  MoveL 1328 to (313.05, 55, -156.48) mm, rotated rx -179.9 ry 0 rz -90 deg; joints [36.817, -66.564, 102.365, -127.219, 48.796, 139.976]
  MoveL 1329 to (313.57, 54.92, -158.6) mm, rotated rx -179.9 ry 0 rz -90 deg; joints [36.783, -66.439, 102.192, -127.22, 48.744, 139.947]
  MoveL 1330 to (314.82, 54.85, -160.4) mm, rotated rx -179.9 ry 0 rz -90 deg; joints [36.779, -66.303, 102.002, -127.186, 48.71, 139.892]
  MoveL 1331 to (316.62, 54.77, -161.63) mm, rotated rx -179.9 ry 0 rz -90 deg; joints [36.807, -66.175, 101.822, -127.121, 48.697, 139.819]
  MoveL 1332 to (318.74, 54.69, -162.14) mm, rotated rx -179.9 ry 0 rz -90 deg; joints [36.863, -66.07, 101.676, -127.036, 48.707, 139.738]
  MoveL 1333 to (320.91, 54.62, -161.86) mm, rotated rx -179.9 ry 0 rz -90 deg; joints [36.938, -66.003, 101.582, -126.941, 48.74, 139.661]
  MoveL 1334 to (322.84, 54.54, -160.83) mm, rotated rx -179.9 ry 0 rz -90 deg; joints [37.023, -65.981, 101.554, -126.851, 48.792, 139.599]
  MoveL 1335 to (324.27, 54.46, -159.18) mm, rotated rx -179.9 ry 0 rz -90 deg; joints [37.108, -66.007, 101.595, -126.776, 48.857, 139.561]
  MoveL 1336 to (325.02, 54.39, -157.13) mm, rotated rx -179.9 ry 0 rz -90 deg; joints [37.181, -66.077, 101.702, -126.728, 48.925, 139.552]
  MoveL 1337 to (324.98, 54.31, -154.94) mm, rotated rx -179.9 ry 0 rz -90 deg; joints [37.232, -66.183, 101.859, -126.712, 48.99, 139.573]
  MoveL 1338 to (324.18, 54.23, -152.91) mm, rotated rx -179.9 ry 0 rz -90 deg; joints [37.256, -66.31, 102.047, -126.731, 49.042, 139.623]
  MoveL 1339 to (322.7, 54.16, -151.3) mm, rotated rx -179.9 ry 0 rz -90 deg; joints [37.248, -66.44, 102.241, -126.783, 49.075, 139.696]
  MoveL 1340 to (320.75, 54.08, -150.32) mm, rotated rx -179.9 ry 0 rz -90 deg; joints [37.21, -66.557, 102.416, -126.862, 49.085, 139.782]
  MoveL 1341 to (318.57, 54, -150.11) mm, rotated rx -179.9 ry 0 rz -90 deg; joints [37.146, -66.646, 102.55, -126.958, 49.071, 139.872]
  MoveL 1342 to (316.46, 53.93, -150.68) mm, rotated rx -179.9 ry 0 rz -90 deg; joints [37.065, -66.693, 102.626, -127.059, 49.036, 139.954]
  MoveL 1343 to (314.7, 53.85, -151.96) mm, rotated rx -179.9 ry 0 rz -90 deg; joints [36.978, -66.692, 102.633, -127.153, 48.984, 140.018]
  MoveL 1344 to (313.5, 53.77, -153.79) mm, rotated rx -179.9 ry 0 rz -90 deg; joints [36.896, -66.644, 102.572, -127.226, 48.923, 140.058]
  MoveL 1345 to (313.04, 53.69, -155.93) mm, rotated rx -179.9 ry 0 rz -90 deg; joints [36.83, -66.554, 102.45, -127.271, 48.862, 140.067]
  MoveL 1346 to (313.37, 53.62, -158.09) mm, rotated rx -179.9 ry 0 rz -90 deg; joints [36.789, -66.434, 102.284, -127.281, 48.807, 140.045]
  MoveL 1347 to (314.44, 53.54, -159.99) mm, rotated rx -179.9 ry 0 rz -90 deg; joints [36.778, -66.299, 102.096, -127.255, 48.768, 139.996]
  MoveL 1348 to (316.12, 53.46, -161.38) mm, rotated rx -179.9 ry 0 rz -90 deg; joints [36.798, -66.168, 101.911, -127.198, 48.749, 139.927]
  MoveL 1349 to (318.19, 53.39, -162.09) mm, rotated rx -179.9 ry 0 rz -90 deg; joints [36.847, -66.056, 101.754, -127.116, 48.753, 139.847]
  MoveL 1350 to (320.38, 53.31, -162.01) mm, rotated rx -179.9 ry 0 rz -90 deg; joints [36.918, -65.978, 101.646, -127.023, 48.781, 139.768]
  MoveL 1351 to (322.39, 53.23, -161.15) mm, rotated rx -179.9 ry 0 rz -90 deg; joints [37.002, -65.944, 101.6, -126.93, 48.828, 139.702]
  MoveL 1352 to (323.96, 53.16, -159.64) mm, rotated rx -179.9 ry 0 rz -90 deg; joints [37.088, -65.958, 101.624, -126.851, 48.89, 139.657]
  MoveL 1353 to (324.9, 53.08, -157.67) mm, rotated rx -179.9 ry 0 rz -90 deg; joints [37.165, -66.018, 101.715, -126.795, 48.959, 139.64]
  MoveL 1354 to (325.07, 53, -155.49) mm, rotated rx -179.9 ry 0 rz -90 deg; joints [37.222, -66.116, 101.861, -126.77, 49.025, 139.654]
  MoveL 1355 to (324.45, 52.93, -153.39) mm, rotated rx -179.9 ry 0 rz -90 deg; joints [37.253, -66.239, 102.044, -126.78, 49.081, 139.697]
  MoveL 1356 to (323.13, 52.85, -151.65) mm, rotated rx -179.9 ry 0 rz -90 deg; joints [37.254, -66.37, 102.239, -126.824, 49.119, 139.764]
  MoveL 1357 to (321.27, 52.77, -150.5) mm, rotated rx -179.9 ry 0 rz -90 deg; joints [37.223, -66.492, 102.421, -126.897, 49.135, 139.848]
  MoveL 1358 to (319.13, 52.7, -150.09) mm, rotated rx -179.9 ry 0 rz -90 deg; joints [37.165, -66.589, 102.567, -126.99, 49.128, 139.938]
  MoveL 1359 to (316.97, 52.62, -150.46) mm, rotated rx -179.9 ry 0 rz -90 deg; joints [37.087, -66.647, 102.659, -127.091, 49.098, 140.023]
  MoveL 1360 to (315.1, 52.54, -151.58) mm, rotated rx -179.9 ry 0 rz -90 deg; joints [37.001, -66.659, 102.684, -127.188, 49.05, 140.093]
  MoveL 1361 to (313.74, 52.47, -153.29) mm, rotated rx -179.9 ry 0 rz -90 deg; joints [36.916, -66.622, 102.639, -127.268, 48.99, 140.139]
  MoveL 1362 to (313.08, 52.39, -155.37) mm, rotated rx -179.9 ry 0 rz -90 deg; joints [36.846, -66.542, 102.531, -127.321, 48.928, 140.156]
  MoveL 1363 to (313.21, 52.31, -157.56) mm, rotated rx -179.9 ry 0 rz -90 deg; joints [36.797, -66.428, 102.375, -127.34, 48.871, 140.142]
  MoveL 1364 to (314.11, 52.24, -159.55) mm, rotated rx -179.9 ry 0 rz -90 deg; joints [36.778, -66.296, 102.19, -127.323, 48.827, 140.099]
  MoveL 1365 to (315.65, 52.16, -161.09) mm, rotated rx -179.9 ry 0 rz -90 deg; joints [36.791, -66.162, 102.002, -127.273, 48.803, 140.034]
  MoveL 1366 to (317.65, 52.08, -161.98) mm, rotated rx -179.9 ry 0 rz -90 deg; joints [36.833, -66.043, 101.836, -127.196, 48.801, 139.956]
  MoveL 1367 to (319.83, 52.01, -162.1) mm, rotated rx -179.9 ry 0 rz -90 deg; joints [36.899, -65.956, 101.713, -127.105, 48.822, 139.876]
  MoveL 1368 to (321.91, 51.93, -161.44) mm, rotated rx -179.9 ry 0 rz -90 deg; joints [36.981, -65.91, 101.651, -127.011, 48.865, 139.805]
  MoveL 1369 to (323.62, 51.85, -160.08) mm, rotated rx -179.9 ry 0 rz -90 deg; joints [37.067, -65.912, 101.658, -126.926, 48.924, 139.754]
  MoveL 1370 to (324.73, 51.78, -158.2) mm, rotated rx -179.9 ry 0 rz -90 deg; joints [37.148, -65.961, 101.732, -126.864, 48.992, 139.729]
  MoveL 1371 to (325.1, 51.7, -156.04) mm, rotated rx -179.9 ry 0 rz -90 deg; joints [37.211, -66.05, 101.866, -126.831, 49.059, 139.735]
  MoveL 1372 to (324.68, 51.62, -153.9) mm, rotated rx -179.9 ry 0 rz -90 deg; joints [37.249, -66.168, 102.041, -126.832, 49.119, 139.772]
  MoveL 1373 to (323.52, 51.55, -152.05) mm, rotated rx -179.9 ry 0 rz -90 deg; joints [37.257, -66.299, 102.235, -126.868, 49.162, 139.834]
  MoveL 1374 to (321.78, 51.47, -150.73) mm, rotated rx -179.9 ry 0 rz -90 deg; joints [37.234, -66.425, 102.423, -126.934, 49.184, 139.914]
  MoveL 1375 to (319.68, 51.39, -150.12) mm, rotated rx -179.9 ry 0 rz -90 deg; joints [37.182, -66.529, 102.581, -127.023, 49.183, 140.004]
  MoveL 1376 to (317.5, 51.32, -150.29) mm, rotated rx -179.9 ry 0 rz -90 deg; joints [37.109, -66.598, 102.687, -127.123, 49.158, 140.091]
  MoveL 1377 to (315.53, 51.24, -151.23) mm, rotated rx -179.9 ry 0 rz -90 deg; joints [37.024, -66.622, 102.73, -127.222, 49.114, 140.165]
  MoveL 1378 to (314.02, 51.16, -152.81) mm, rotated rx -179.9 ry 0 rz -90 deg; joints [36.938, -66.597, 102.702, -127.307, 49.057, 140.218]
  MoveL 1379 to (313.18, 51.09, -154.83) mm, rotated rx -179.9 ry 0 rz -90 deg; joints [36.862, -66.528, 102.61, -127.368, 48.995, 140.243]
  MoveL 1380 to (313.1, 51.01, -157.01) mm, rotated rx -179.9 ry 0 rz -90 deg; joints [36.808, -66.421, 102.463, -127.396, 48.936, 140.236]
  MoveL 1381 to (313.81, 50.93, -159.08) mm, rotated rx -179.9 ry 0 rz -90 deg; joints [36.781, -66.292, 102.284, -127.388, 48.888, 140.2]
  MoveL 1382 to (315.21, 50.86, -160.76) mm, rotated rx -179.9 ry 0 rz -90 deg; joints [36.785, -66.157, 102.094, -127.346, 48.858, 140.14]
  MoveL 1383 to (317.12, 50.78, -161.83) mm, rotated rx -179.9 ry 0 rz -90 deg; joints [36.82, -66.033, 101.92, -127.275, 48.85, 140.064]
  MoveL 1384 to (319.28, 50.7, -162.15) mm, rotated rx -179.9 ry 0 rz -90 deg; joints [36.881, -65.936, 101.785, -127.186, 48.866, 139.983]
  MoveL 1385 to (321.41, 50.63, -161.68) mm, rotated rx -179.9 ry 0 rz -90 deg; joints [36.96, -65.879, 101.706, -127.091, 48.904, 139.909]
  MoveL 1386 to (323.24, 50.55, -160.48) mm, rotated rx -179.9 ry 0 rz -90 deg; joints [37.046, -65.869, 101.695, -127.004, 48.959, 139.852]
  MoveL 1387 to (324.52, 50.47, -158.71) mm, rotated rx -179.9 ry 0 rz -90 deg; joints [37.129, -65.907, 101.753, -126.934, 49.025, 139.821]
  MoveL 1388 to (325.08, 50.4, -156.59) mm, rotated rx -179.9 ry 0 rz -90 deg; joints [37.198, -65.987, 101.873, -126.893, 49.093, 139.819]
  MoveL 1389 to (324.86, 50.32, -154.42) mm, rotated rx -179.9 ry 0 rz -90 deg; joints [37.243, -66.099, 102.04, -126.885, 49.156, 139.848]
  MoveL 1390 to (323.87, 50.24, -152.47) mm, rotated rx -179.9 ry 0 rz -90 deg; joints [37.259, -66.228, 102.232, -126.913, 49.204, 139.904]
  MoveL 1391 to (322.26, 50.17, -151) mm, rotated rx -179.9 ry 0 rz -90 deg; joints [37.243, -66.356, 102.424, -126.972, 49.232, 139.981]
  MoveL 1392 to (320.23, 50.09, -150.2) mm, rotated rx -179.9 ry 0 rz -90 deg; joints [37.198, -66.467, 102.591, -127.056, 49.236, 140.069]
  MoveL 1393 to (318.04, 50.01, -150.17) mm, rotated rx -179.9 ry 0 rz -90 deg; joints [37.13, -66.546, 102.712, -127.154, 49.218, 140.158]
  MoveL 1394 to (315.99, 49.94, -150.93) mm, rotated rx -179.9 ry 0 rz -90 deg; joints [37.046, -66.582, 102.771, -127.255, 49.178, 140.236]
  MoveL 1395 to (314.35, 49.86, -152.36) mm, rotated rx -179.9 ry 0 rz -90 deg; joints [36.959, -66.57, 102.761, -127.345, 49.124, 140.295]
  MoveL 1396 to (313.32, 49.78, -154.29) mm, rotated rx -179.9 ry 0 rz -90 deg; joints [36.88, -66.511, 102.684, -127.413, 49.062, 140.327]
  MoveL 1397 to (313.05, 49.71, -156.46) mm, rotated rx -179.9 ry 0 rz -90 deg; joints [36.82, -66.412, 102.55, -127.449, 49.002, 140.329]
  MoveL 1398 to (313.56, 49.63, -158.58) mm, rotated rx -179.9 ry 0 rz -90 deg; joints [36.785, -66.287, 102.376, -127.451, 48.95, 140.3]
  MoveL 1399 to (314.8, 49.55, -160.38) mm, rotated rx -179.9 ry 0 rz -90 deg; joints [36.782, -66.152, 102.187, -127.417, 48.915, 140.245]
  MoveL 1400 to (316.6, 49.48, -161.62) mm, rotated rx -179.9 ry 0 rz -90 deg; joints [36.81, -66.024, 102.007, -127.352, 48.901, 140.172]
  MoveL 1401 to (318.72, 49.4, -162.14) mm, rotated rx -179.9 ry 0 rz -90 deg; joints [36.865, -65.919, 101.86, -127.267, 48.911, 140.091]
  MoveL 1402 to (320.89, 49.32, -161.87) mm, rotated rx -179.9 ry 0 rz -90 deg; joints [36.94, -65.851, 101.765, -127.173, 48.943, 140.015]
  MoveL 1403 to (322.82, 49.25, -160.84) mm, rotated rx -179.9 ry 0 rz -90 deg; joints [37.025, -65.829, 101.737, -127.082, 48.994, 139.953]
  MoveL 1404 to (324.26, 49.17, -159.19) mm, rotated rx -179.9 ry 0 rz -90 deg; joints [37.11, -65.855, 101.778, -127.007, 49.058, 139.914]
  MoveL 1405 to (325.01, 49.09, -157.14) mm, rotated rx -179.9 ry 0 rz -90 deg; joints [37.183, -65.925, 101.883, -126.958, 49.127, 139.905]
  MoveL 1406 to (324.99, 49.01, -154.96) mm, rotated rx -179.9 ry 0 rz -90 deg; joints [37.235, -66.03, 102.04, -126.941, 49.192, 139.926]
  MoveL 1407 to (324.19, 48.94, -152.93) mm, rotated rx -179.9 ry 0 rz -90 deg; joints [37.258, -66.156, 102.228, -126.96, 49.244, 139.976]
  MoveL 1408 to (322.72, 48.86, -151.31) mm, rotated rx -179.9 ry 0 rz -90 deg; joints [37.251, -66.286, 102.422, -127.011, 49.278, 140.048]
  MoveL 1409 to (320.76, 48.78, -150.33) mm, rotated rx -179.9 ry 0 rz -90 deg; joints [37.213, -66.403, 102.598, -127.09, 49.288, 140.134]
  MoveL 1410 to (318.59, 48.71, -150.1) mm, rotated rx -179.9 ry 0 rz -90 deg; joints [37.149, -66.492, 102.732, -127.186, 49.276, 140.224]
  MoveL 1411 to (316.48, 48.63, -150.67) mm, rotated rx -179.9 ry 0 rz -90 deg; joints [37.069, -66.539, 102.808, -127.287, 49.241, 140.306]
  MoveL 1412 to (314.71, 48.55, -151.95) mm, rotated rx -179.9 ry 0 rz -90 deg; joints [36.982, -66.539, 102.816, -127.381, 49.19, 140.37]
  MoveL 1413 to (313.51, 48.48, -153.77) mm, rotated rx -179.9 ry 0 rz -90 deg; joints [36.9, -66.491, 102.755, -127.455, 49.13, 140.41]
  MoveL 1414 to (313.04, 48.4, -155.91) mm, rotated rx -179.9 ry 0 rz -90 deg; joints [36.833, -66.402, 102.634, -127.5, 49.068, 140.419]
  MoveL 1415 to (313.36, 48.32, -158.07) mm, rotated rx -179.9 ry 0 rz -90 deg; joints [36.792, -66.282, 102.468, -127.511, 49.013, 140.398]
  MoveL 1416 to (314.43, 48.25, -159.97) mm, rotated rx -179.9 ry 0 rz -90 deg; joints [36.781, -66.148, 102.28, -127.485, 48.973, 140.349]
  MoveL 1417 to (316.11, 48.17, -161.37) mm, rotated rx -179.9 ry 0 rz -90 deg; joints [36.801, -66.016, 102.095, -127.428, 48.954, 140.279]
  MoveL 1418 to (318.17, 48.09, -162.08) mm, rotated rx -179.9 ry 0 rz -90 deg; joints [36.849, -65.904, 101.938, -127.347, 48.957, 140.2]
  MoveL 1419 to (320.36, 48.02, -162.01) mm, rotated rx -179.9 ry 0 rz -90 deg; joints [36.92, -65.826, 101.829, -127.254, 48.984, 140.121]
  MoveL 1420 to (322.37, 47.94, -161.17) mm, rotated rx -179.9 ry 0 rz -90 deg; joints [37.004, -65.792, 101.783, -127.161, 49.031, 140.054]
  MoveL 1421 to (323.95, 47.86, -159.66) mm, rotated rx -179.9 ry 0 rz -90 deg; joints [37.09, -65.806, 101.806, -127.081, 49.092, 140.009]
  MoveL 1422 to (324.89, 47.79, -157.69) mm, rotated rx -179.9 ry 0 rz -90 deg; joints [37.167, -65.865, 101.896, -127.024, 49.161, 139.992]
  MoveL 1423 to (325.07, 47.71, -155.51) mm, rotated rx -179.9 ry 0 rz -90 deg; joints [37.225, -65.963, 102.042, -126.999, 49.227, 140.006]
  MoveL 1424 to (324.46, 47.63, -153.41) mm, rotated rx -179.9 ry 0 rz -90 deg; joints [37.256, -66.085, 102.224, -127.009, 49.283, 140.049]
  MoveL 1425 to (323.14, 47.56, -151.67) mm, rotated rx -179.9 ry 0 rz -90 deg; joints [37.256, -66.216, 102.419, -127.052, 49.322, 140.116]
  MoveL 1426 to (321.29, 47.48, -150.51) mm, rotated rx -179.9 ry 0 rz -90 deg; joints [37.226, -66.337, 102.602, -127.125, 49.339, 140.2]
  MoveL 1427 to (319.14, 47.4, -150.09) mm, rotated rx -179.9 ry 0 rz -90 deg; joints [37.168, -66.434, 102.749, -127.218, 49.332, 140.289]
  MoveL 1428 to (316.99, 47.33, -150.45) mm, rotated rx -179.9 ry 0 rz -90 deg; joints [37.091, -66.493, 102.84, -127.319, 49.303, 140.374]
  MoveL 1429 to (315.11, 47.25, -151.57) mm, rotated rx -179.9 ry 0 rz -90 deg; joints [37.004, -66.505, 102.866, -127.416, 49.256, 140.444]
  MoveL 1430 to (313.75, 47.17, -153.27) mm, rotated rx -179.9 ry 0 rz -90 deg; joints [36.92, -66.469, 102.822, -127.496, 49.197, 140.49]
  MoveL 1431 to (313.08, 47.1, -155.36) mm, rotated rx -179.9 ry 0 rz -90 deg; joints [36.849, -66.389, 102.715, -127.549, 49.135, 140.507]
  MoveL 1432 to (313.2, 47.02, -157.54) mm, rotated rx -179.9 ry 0 rz -90 deg; joints [36.8, -66.276, 102.558, -127.569, 49.077, 140.493]
  MoveL 1433 to (314.1, 46.94, -159.53) mm, rotated rx -179.9 ry 0 rz -90 deg; joints [36.781, -66.144, 102.374, -127.552, 49.033, 140.451]
  MoveL 1434 to (315.64, 46.87, -161.08) mm, rotated rx -179.9 ry 0 rz -90 deg; joints [36.793, -66.01, 102.186, -127.502, 49.008, 140.386]
  MoveL 1435 to (317.63, 46.79, -161.98) mm, rotated rx -179.9 ry 0 rz -90 deg; joints [36.835, -65.892, 102.019, -127.426, 49.005, 140.308]
  MoveL 1436 to (319.81, 46.71, -162.1) mm, rotated rx -179.9 ry 0 rz -90 deg; joints [36.901, -65.804, 101.896, -127.335, 49.026, 140.228]
  MoveL 1437 to (321.89, 46.64, -161.45) mm, rotated rx -179.9 ry 0 rz -90 deg; joints [36.983, -65.758, 101.833, -127.241, 49.068, 140.157]
  MoveL 1438 to (323.61, 46.56, -160.09) mm, rotated rx -179.9 ry 0 rz -90 deg; joints [37.069, -65.759, 101.839, -127.156, 49.127, 140.106]
  MoveL 1439 to (324.73, 46.48, -158.21) mm, rotated rx -179.9 ry 0 rz -90 deg; joints [37.15, -65.808, 101.913, -127.093, 49.194, 140.081]
  MoveL 1440 to (325.1, 46.41, -156.06) mm, rotated rx -179.9 ry 0 rz -90 deg; joints [37.213, -65.897, 102.046, -127.059, 49.262, 140.087]
  MoveL 1441 to (324.68, 46.33, -153.92) mm, rotated rx -179.9 ry 0 rz -90 deg; joints [37.252, -66.014, 102.221, -127.06, 49.321, 140.123]
  MoveL 1442 to (323.53, 46.25, -152.06) mm, rotated rx -179.9 ry 0 rz -90 deg; joints [37.26, -66.144, 102.415, -127.095, 49.365, 140.185]
  MoveL 1443 to (321.79, 46.18, -150.74) mm, rotated rx -179.9 ry 0 rz -90 deg; joints [37.237, -66.27, 102.603, -127.161, 49.388, 140.265]
  MoveL 1444 to (319.7, 46.1, -150.12) mm, rotated rx -179.9 ry 0 rz -90 deg; joints [37.186, -66.374, 102.761, -127.25, 49.387, 140.354]
  MoveL 1445 to (317.52, 46.02, -150.29) mm, rotated rx -179.9 ry 0 rz -90 deg; joints [37.112, -66.443, 102.868, -127.35, 49.364, 140.441]
  MoveL 1446 to (315.54, 45.95, -151.22) mm, rotated rx -179.9 ry 0 rz -90 deg; joints [37.027, -66.467, 102.911, -127.449, 49.32, 140.516]
  MoveL 1447 to (314.03, 45.87, -152.8) mm, rotated rx -179.9 ry 0 rz -90 deg; joints [36.941, -66.443, 102.885, -127.535, 49.264, 140.569]
  MoveL 1448 to (313.18, 45.79, -154.81) mm, rotated rx -179.9 ry 0 rz -90 deg; joints [36.866, -66.374, 102.792, -127.595, 49.202, 140.593]
  MoveL 1449 to (313.1, 45.72, -156.99) mm, rotated rx -179.9 ry 0 rz -90 deg; joints [36.811, -66.268, 102.646, -127.624, 49.142, 140.587]
  MoveL 1450 to (313.8, 45.64, -159.06) mm, rotated rx -179.9 ry 0 rz -90 deg; joints [36.784, -66.139, 102.467, -127.617, 49.094, 140.551]
  MoveL 1451 to (315.2, 45.56, -160.74) mm, rotated rx -179.9 ry 0 rz -90 deg; joints [36.788, -66.004, 102.277, -127.575, 49.063, 140.491]
  MoveL 1452 to (317.1, 45.49, -161.82) mm, rotated rx -179.9 ry 0 rz -90 deg; joints [36.823, -65.881, 102.103, -127.504, 49.055, 140.415]
  MoveL 1453 to (319.26, 45.41, -162.15) mm, rotated rx -179.9 ry 0 rz -90 deg; joints [36.883, -65.784, 101.967, -127.416, 49.07, 140.335]
  MoveL 1454 to (321.39, 45.33, -161.68) mm, rotated rx -179.9 ry 0 rz -90 deg; joints [36.962, -65.727, 101.888, -127.321, 49.107, 140.261]
  MoveL 1455 to (323.22, 45.26, -160.49) mm, rotated rx -179.9 ry 0 rz -90 deg; joints [37.048, -65.716, 101.876, -127.233, 49.162, 140.204]
  MoveL 1456 to (324.51, 45.18, -158.72) mm, rotated rx -179.9 ry 0 rz -90 deg; joints [37.131, -65.753, 101.933, -127.163, 49.227, 140.172]
  MoveL 1457 to (325.08, 45.1, -156.61) mm, rotated rx -179.9 ry 0 rz -90 deg; joints [37.2, -65.833, 102.053, -127.121, 49.296, 140.17]
  MoveL 1458 to (324.86, 45.03, -154.44) mm, rotated rx -179.9 ry 0 rz -90 deg; joints [37.245, -65.944, 102.219, -127.113, 49.358, 140.199]
  MoveL 1459 to (323.89, 44.95, -152.49) mm, rotated rx -179.9 ry 0 rz -90 deg; joints [37.262, -66.072, 102.411, -127.14, 49.407, 140.255]
  MoveL 1460 to (322.28, 44.87, -151.01) mm, rotated rx -179.9 ry 0 rz -90 deg; joints [37.246, -66.201, 102.603, -127.199, 49.435, 140.331]
  MoveL 1461 to (320.25, 44.8, -150.2) mm, rotated rx -179.9 ry 0 rz -90 deg; joints [37.202, -66.312, 102.771, -127.282, 49.441, 140.419]
  MoveL 1462 to (318.06, 44.72, -150.17) mm, rotated rx -179.9 ry 0 rz -90 deg; joints [37.133, -66.391, 102.892, -127.381, 49.423, 140.508]
  MoveL 1463 to (316.01, 44.64, -150.92) mm, rotated rx -179.9 ry 0 rz -90 deg; joints [37.05, -66.427, 102.952, -127.481, 49.384, 140.586]
  MoveL 1464 to (314.36, 44.56, -152.35) mm, rotated rx -179.9 ry 0 rz -90 deg; joints [36.963, -66.415, 102.943, -127.571, 49.331, 140.645]
  MoveL 1465 to (313.32, 44.49, -154.27) mm, rotated rx -179.9 ry 0 rz -90 deg; joints [36.884, -66.356, 102.866, -127.64, 49.269, 140.677]
  MoveL 1466 to (313.04, 44.41, -156.44) mm, rotated rx -179.9 ry 0 rz -90 deg; joints [36.823, -66.259, 102.732, -127.677, 49.208, 140.679]
  MoveL 1467 to (313.56, 44.33, -158.57) mm, rotated rx -179.9 ry 0 rz -90 deg; joints [36.788, -66.134, 102.559, -127.678, 49.156, 140.65]
  MoveL 1468 to (314.79, 44.26, -160.37) mm, rotated rx -179.9 ry 0 rz -90 deg; joints [36.785, -65.999, 102.369, -127.645, 49.121, 140.596]
  MoveL 1469 to (316.58, 44.18, -161.61) mm, rotated rx -179.9 ry 0 rz -90 deg; joints [36.812, -65.871, 102.189, -127.581, 49.106, 140.523]
  MoveL 1470 to (318.71, 44.1, -162.14) mm, rotated rx -179.9 ry 0 rz -90 deg; joints [36.867, -65.767, 102.041, -127.496, 49.115, 140.442]
  MoveL 1471 to (320.87, 44.03, -161.87) mm, rotated rx -179.9 ry 0 rz -90 deg; joints [36.942, -65.699, 101.946, -127.401, 49.147, 140.365]
  MoveL 1472 to (322.81, 43.95, -160.85) mm, rotated rx -179.9 ry 0 rz -90 deg; joints [37.027, -65.676, 101.917, -127.31, 49.197, 140.303]
  MoveL 1473 to (324.25, 43.87, -159.21) mm, rotated rx -179.9 ry 0 rz -90 deg; joints [37.112, -65.701, 101.957, -127.235, 49.261, 140.265]
  MoveL 1474 to (325.01, 43.8, -157.16) mm, rotated rx -179.9 ry 0 rz -90 deg; joints [37.185, -65.771, 102.063, -127.185, 49.33, 140.255]
  MoveL 1475 to (324.99, 43.72, -154.98) mm, rotated rx -179.9 ry 0 rz -90 deg; joints [37.237, -65.875, 102.219, -127.168, 49.394, 140.276]
  MoveL 1476 to (324.2, 43.64, -152.94) mm, rotated rx -179.9 ry 0 rz -90 deg; joints [37.261, -66.001, 102.407, -127.186, 49.447, 140.326]
  MoveL 1477 to (322.73, 43.57, -151.32) mm, rotated rx -179.9 ry 0 rz -90 deg; joints [37.254, -66.131, 102.601, -127.237, 49.481, 140.398]
  MoveL 1478 to (320.78, 43.49, -150.33) mm, rotated rx -179.9 ry 0 rz -90 deg; joints [37.216, -66.247, 102.777, -127.316, 49.493, 140.484]
  MoveL 1479 to (318.61, 43.41, -150.1) mm, rotated rx -179.9 ry 0 rz -90 deg; joints [37.153, -66.336, 102.912, -127.411, 49.481, 140.573]
  MoveL 1480 to (316.5, 43.34, -150.66) mm, rotated rx -179.9 ry 0 rz -90 deg; joints [37.072, -66.383, 102.988, -127.513, 49.447, 140.655]
  MoveL 1481 to (314.72, 43.26, -151.93) mm, rotated rx -179.9 ry 0 rz -90 deg; joints [36.985, -66.384, 102.997, -127.607, 49.397, 140.72]
  MoveL 1482 to (313.52, 43.18, -153.76) mm, rotated rx -179.9 ry 0 rz -90 deg; joints [36.903, -66.336, 102.936, -127.681, 49.337, 140.759]
  MoveL 1483 to (313.04, 43.11, -155.89) mm, rotated rx -179.9 ry 0 rz -90 deg; joints [36.837, -66.247, 102.815, -127.727, 49.275, 140.769]
  MoveL 1484 to (313.35, 43.03, -158.05) mm, rotated rx -179.9 ry 0 rz -90 deg; joints [36.795, -66.128, 102.65, -127.738, 49.22, 140.747]
  MoveL 1485 to (314.42, 42.95, -159.96) mm, rotated rx -179.9 ry 0 rz -90 deg; joints [36.783, -65.994, 102.462, -127.713, 49.18, 140.699]
  MoveL 1486 to (316.09, 42.88, -161.36) mm, rotated rx -179.9 ry 0 rz -90 deg; joints [36.803, -65.863, 102.277, -127.656, 49.159, 140.629]
  MoveL 1487 to (318.15, 42.8, -162.08) mm, rotated rx -179.9 ry 0 rz -90 deg; joints [36.851, -65.751, 102.119, -127.575, 49.162, 140.55]
  MoveL 1488 to (320.34, 42.72, -162.01) mm, rotated rx -179.9 ry 0 rz -90 deg; joints [36.922, -65.673, 102.009, -127.482, 49.188, 140.471]
  MoveL 1489 to (322.36, 42.65, -161.18) mm, rotated rx -179.9 ry 0 rz -90 deg; joints [37.006, -65.638, 101.963, -127.389, 49.234, 140.404]
  MoveL 1490 to (323.94, 42.57, -159.67) mm, rotated rx -179.9 ry 0 rz -90 deg; joints [37.092, -65.652, 101.986, -127.308, 49.295, 140.359]
  MoveL 1491 to (324.89, 42.49, -157.7) mm, rotated rx -179.9 ry 0 rz -90 deg; joints [37.169, -65.711, 102.075, -127.251, 49.363, 140.342]
  MoveL 1492 to (325.07, 42.42, -155.53) mm, rotated rx -179.9 ry 0 rz -90 deg; joints [37.227, -65.807, 102.221, -127.226, 49.43, 140.355]
  MoveL 1493 to (324.47, 42.34, -153.43) mm, rotated rx -179.9 ry 0 rz -90 deg; joints [37.259, -65.929, 102.402, -127.235, 49.486, 140.398]
  MoveL 1494 to (323.15, 42.26, -151.68) mm, rotated rx -179.9 ry 0 rz -90 deg; joints [37.259, -66.059, 102.597, -127.278, 49.526, 140.465]
  MoveL 1495 to (321.31, 42.19, -150.52) mm, rotated rx -179.9 ry 0 rz -90 deg; joints [37.229, -66.181, 102.78, -127.35, 49.544, 140.548]
  MoveL 1496 to (319.16, 42.11, -150.09) mm, rotated rx -179.9 ry 0 rz -90 deg; joints [37.171, -66.278, 102.927, -127.442, 49.538, 140.638]
  MoveL 1497 to (317.01, 42.03, -150.45) mm, rotated rx -179.9 ry 0 rz -90 deg; joints [37.094, -66.336, 103.02, -127.544, 49.509, 140.723]
  MoveL 1498 to (315.12, 41.96, -151.55) mm, rotated rx -179.9 ry 0 rz -90 deg; joints [37.008, -66.349, 103.046, -127.641, 49.462, 140.793]
  MoveL 1499 to (313.76, 41.88, -153.26) mm, rotated rx -179.9 ry 0 rz -90 deg; joints [36.923, -66.313, 103.002, -127.721, 49.404, 140.839]
  MoveL 1500 to (313.09, 41.8, -155.34) mm, rotated rx -179.9 ry 0 rz -90 deg; joints [36.852, -66.234, 102.895, -127.775, 49.342, 140.856]
  MoveL 1501 to (313.2, 41.73, -157.52) mm, rotated rx -179.9 ry 0 rz -90 deg; joints [36.803, -66.121, 102.739, -127.795, 49.284, 140.842]
  MoveL 1502 to (314.08, 41.65, -159.52) mm, rotated rx -179.9 ry 0 rz -90 deg; joints [36.784, -65.99, 102.555, -127.779, 49.24, 140.8]
  MoveL 1503 to (315.62, 41.57, -161.07) mm, rotated rx -179.9 ry 0 rz -90 deg; joints [36.796, -65.856, 102.367, -127.73, 49.214, 140.735]
  MoveL 1504 to (317.61, 41.5, -161.97) mm, rotated rx -179.9 ry 0 rz -90 deg; joints [36.837, -65.738, 102.2, -127.654, 49.21, 140.657]
  MoveL 1505 to (319.79, 41.42, -162.11) mm, rotated rx -179.9 ry 0 rz -90 deg; joints [36.903, -65.65, 102.076, -127.562, 49.231, 140.577]
  MoveL 1506 to (321.88, 41.34, -161.46) mm, rotated rx -179.9 ry 0 rz -90 deg; joints [36.985, -65.604, 102.013, -127.468, 49.272, 140.506]
  MoveL 1507 to (323.6, 41.27, -160.1) mm, rotated rx -179.9 ry 0 rz -90 deg; joints [37.071, -65.605, 102.018, -127.383, 49.33, 140.455]
  MoveL 1508 to (324.72, 41.19, -158.23) mm, rotated rx -179.9 ry 0 rz -90 deg; joints [37.152, -65.653, 102.092, -127.319, 49.397, 140.43]
  MoveL 1509 to (325.1, 41.11, -156.08) mm, rotated rx -179.9 ry 0 rz -90 deg; joints [37.215, -65.741, 102.224, -127.285, 49.465, 140.436]
  MoveL 1510 to (324.69, 41.04, -153.93) mm, rotated rx -179.9 ry 0 rz -90 deg; joints [37.254, -65.858, 102.399, -127.285, 49.525, 140.472]
  MoveL 1511 to (323.54, 40.96, -152.07) mm, rotated rx -179.9 ry 0 rz -90 deg; joints [37.263, -65.988, 102.593, -127.32, 49.569, 140.533]
  MoveL 1512 to (321.81, 40.88, -150.74) mm, rotated rx -179.9 ry 0 rz -90 deg; joints [37.24, -66.113, 102.781, -127.386, 49.593, 140.613]
  MoveL 1513 to (319.72, 40.81, -150.12) mm, rotated rx -179.9 ry 0 rz -90 deg; joints [37.189, -66.217, 102.939, -127.474, 49.593, 140.702]
  MoveL 1514 to (317.54, 40.73, -150.28) mm, rotated rx -179.9 ry 0 rz -90 deg; joints [37.116, -66.286, 103.047, -127.574, 49.57, 140.789]
  MoveL 1515 to (315.56, 40.65, -151.21) mm, rotated rx -179.9 ry 0 rz -90 deg; joints [37.03, -66.311, 103.09, -127.673, 49.527, 140.864]
  MoveL 1516 to (314.04, 40.58, -152.78) mm, rotated rx -179.9 ry 0 rz -90 deg; joints [36.944, -66.287, 103.064, -127.759, 49.471, 140.917]
  MoveL 1517 to (313.18, 40.5, -154.79) mm, rotated rx -179.9 ry 0 rz -90 deg; joints [36.869, -66.218, 102.972, -127.821, 49.409, 140.942]
  MoveL 1518 to (313.1, 40.42, -156.97) mm, rotated rx -179.9 ry 0 rz -90 deg; joints [36.814, -66.113, 102.827, -127.85, 49.35, 140.936]
  MoveL 1519 to (313.79, 40.35, -159.04) mm, rotated rx -179.9 ry 0 rz -90 deg; joints [36.787, -65.985, 102.647, -127.843, 49.301, 140.9]
  MoveL 1520 to (315.18, 40.27, -160.73) mm, rotated rx -179.9 ry 0 rz -90 deg; joints [36.79, -65.85, 102.458, -127.801, 49.27, 140.84]
  MoveL 1521 to (317.08, 40.19, -161.81) mm, rotated rx -179.9 ry 0 rz -90 deg; joints [36.825, -65.726, 102.283, -127.731, 49.26, 140.764]
  MoveL 1522 to (319.24, 40.12, -162.15) mm, rotated rx -179.9 ry 0 rz -90 deg; joints [36.885, -65.63, 102.147, -127.643, 49.275, 140.684]
  MoveL 1523 to (321.38, 40.04, -161.69) mm, rotated rx -179.9 ry 0 rz -90 deg; joints [36.964, -65.572, 102.067, -127.547, 49.311, 140.609]
  MoveL 1524 to (323.21, 39.96, -160.5) mm, rotated rx -179.9 ry 0 rz -90 deg; joints [37.05, -65.561, 102.054, -127.459, 49.365, 140.552]
  MoveL 1525 to (324.5, 39.88, -158.74) mm, rotated rx -179.9 ry 0 rz -90 deg; joints [37.133, -65.598, 102.111, -127.389, 49.431, 140.52]
  MoveL 1526 to (325.08, 39.81, -156.63) mm, rotated rx -179.9 ry 0 rz -90 deg; joints [37.202, -65.677, 102.231, -127.347, 49.499, 140.518]
  MoveL 1527 to (324.87, 39.73, -154.46) mm, rotated rx -179.9 ry 0 rz -90 deg; joints [37.248, -65.788, 102.397, -127.338, 49.562, 140.547]
  MoveL 1528 to (323.9, 39.65, -152.5) mm, rotated rx -179.9 ry 0 rz -90 deg; joints [37.264, -65.916, 102.588, -127.364, 49.611, 140.603]
  MoveL 1529 to (322.29, 39.58, -151.02) mm, rotated rx -179.9 ry 0 rz -90 deg; joints [37.249, -66.044, 102.78, -127.422, 49.64, 140.679]
  MoveL 1530 to (320.26, 39.5, -150.2) mm, rotated rx -179.9 ry 0 rz -90 deg; joints [37.205, -66.155, 102.948, -127.506, 49.646, 140.767]
  MoveL 1531 to (318.08, 39.42, -150.17) mm, rotated rx -179.9 ry 0 rz -90 deg; joints [37.136, -66.234, 103.07, -127.604, 49.629, 140.855]
  MoveL 1532 to (316.02, 39.35, -150.91) mm, rotated rx -179.9 ry 0 rz -90 deg; joints [37.053, -66.27, 103.131, -127.705, 49.591, 140.934]
  MoveL 1533 to (314.37, 39.27, -152.33) mm, rotated rx -179.9 ry 0 rz -90 deg; joints [36.966, -66.258, 103.122, -127.795, 49.538, 140.993]
  MoveL 1534 to (313.33, 39.19, -154.26) mm, rotated rx -179.9 ry 0 rz -90 deg; joints [36.887, -66.2, 103.046, -127.864, 49.477, 141.025]
  MoveL 1535 to (313.04, 39.12, -156.42) mm, rotated rx -179.9 ry 0 rz -90 deg; joints [36.826, -66.103, 102.912, -127.902, 49.416, 141.027]
  MoveL 1536 to (313.55, 39.04, -158.55) mm, rotated rx -179.9 ry 0 rz -90 deg; joints [36.791, -65.979, 102.739, -127.904, 49.364, 140.998]
  MoveL 1537 to (314.78, 38.96, -160.36) mm, rotated rx -179.9 ry 0 rz -90 deg; joints [36.787, -65.844, 102.549, -127.871, 49.327, 140.944]
  MoveL 1538 to (316.57, 38.89, -161.61) mm, rotated rx -179.9 ry 0 rz -90 deg; joints [36.814, -65.717, 102.369, -127.807, 49.312, 140.871]
  MoveL 1539 to (318.69, 38.81, -162.14) mm, rotated rx -179.9 ry 0 rz -90 deg; joints [36.869, -65.612, 102.221, -127.722, 49.32, 140.79]
  MoveL 1540 to (320.86, 38.73, -161.88) mm, rotated rx -179.9 ry 0 rz -90 deg; joints [36.944, -65.544, 102.125, -127.627, 49.351, 140.714]
  MoveL 1541 to (322.79, 38.66, -160.86) mm, rotated rx -179.9 ry 0 rz -90 deg; joints [37.029, -65.521, 102.095, -127.536, 49.401, 140.651]
  MoveL 1542 to (324.24, 38.58, -159.23) mm, rotated rx -179.9 ry 0 rz -90 deg; joints [37.114, -65.545, 102.135, -127.46, 49.465, 140.612]
  MoveL 1543 to (325.01, 38.5, -157.18) mm, rotated rx -179.9 ry 0 rz -90 deg; joints [37.187, -65.614, 102.24, -127.41, 49.533, 140.603]
  MoveL 1544 to (325, 38.43, -155) mm, rotated rx -179.9 ry 0 rz -90 deg; joints [37.239, -65.718, 102.396, -127.392, 49.598, 140.624]
  MoveL 1545 to (324.21, 38.35, -152.96) mm, rotated rx -179.9 ry 0 rz -90 deg; joints [37.264, -65.843, 102.583, -127.41, 49.651, 140.673]
  MoveL 1546 to (322.75, 38.27, -151.34) mm, rotated rx -179.9 ry 0 rz -90 deg; joints [37.257, -65.973, 102.777, -127.461, 49.686, 140.745]
  MoveL 1547 to (320.8, 38.2, -150.34) mm, rotated rx -179.9 ry 0 rz -90 deg; joints [37.219, -66.09, 102.954, -127.539, 49.698, 140.831]
  MoveL 1548 to (318.63, 38.12, -150.1) mm, rotated rx -179.9 ry 0 rz -90 deg; joints [37.156, -66.178, 103.089, -127.634, 49.687, 140.92]
  MoveL 1549 to (316.51, 38.04, -150.65) mm, rotated rx -179.9 ry 0 rz -90 deg; joints [37.076, -66.226, 103.166, -127.736, 49.654, 141.002]
  MoveL 1550 to (314.74, 37.97, -151.92) mm, rotated rx -179.9 ry 0 rz -90 deg; joints [36.988, -66.226, 103.175, -127.83, 49.604, 141.067]
  MoveL 1551 to (313.52, 37.89, -153.74) mm, rotated rx -179.9 ry 0 rz -90 deg; joints [36.906, -66.18, 103.115, -127.905, 49.544, 141.106]
  MoveL 1552 to (313.04, 37.81, -155.87) mm, rotated rx -179.9 ry 0 rz -90 deg; joints [36.84, -66.091, 102.995, -127.951, 49.483, 141.116]
  MoveL 1553 to (313.35, 37.74, -158.03) mm, rotated rx -179.9 ry 0 rz -90 deg; joints [36.798, -65.973, 102.829, -127.963, 49.428, 141.094]
  MoveL 1554 to (314.4, 37.66, -159.94) mm, rotated rx -179.9 ry 0 rz -90 deg; joints [36.786, -65.839, 102.642, -127.938, 49.387, 141.046]
  MoveL 1555 to (316.07, 37.58, -161.35) mm, rotated rx -179.9 ry 0 rz -90 deg; joints [36.805, -65.708, 102.456, -127.882, 49.366, 140.977]
  MoveL 1556 to (318.14, 37.51, -162.08) mm, rotated rx -179.9 ry 0 rz -90 deg; joints [36.853, -65.596, 102.298, -127.801, 49.368, 140.897]
  MoveL 1557 to (320.32, 37.43, -162.02) mm, rotated rx -179.9 ry 0 rz -90 deg; joints [36.924, -65.518, 102.188, -127.707, 49.393, 140.818]
  MoveL 1558 to (322.34, 37.35, -161.19) mm, rotated rx -179.9 ry 0 rz -90 deg; joints [37.008, -65.483, 102.141, -127.614, 49.438, 140.752]
  MoveL 1559 to (323.93, 37.28, -159.69) mm, rotated rx -179.9 ry 0 rz -90 deg; joints [37.094, -65.496, 102.163, -127.533, 49.499, 140.706]
  MoveL 1560 to (324.88, 37.2, -157.72) mm, rotated rx -179.9 ry 0 rz -90 deg; joints [37.171, -65.554, 102.252, -127.476, 49.567, 140.689]
  MoveL 1561 to (325.07, 37.12, -155.55) mm, rotated rx -179.9 ry 0 rz -90 deg; joints [37.229, -65.65, 102.397, -127.449, 49.634, 140.702]
  MoveL 1562 to (324.48, 37.05, -153.44) mm, rotated rx -179.9 ry 0 rz -90 deg; joints [37.261, -65.771, 102.578, -127.458, 49.69, 140.745]
  MoveL 1563 to (323.17, 36.97, -151.69) mm, rotated rx -179.9 ry 0 rz -90 deg; joints [37.262, -65.901, 102.773, -127.501, 49.731, 140.812]
  MoveL 1564 to (321.32, 36.89, -150.52) mm, rotated rx -179.9 ry 0 rz -90 deg; joints [37.232, -66.023, 102.956, -127.573, 49.749, 140.895]
  MoveL 1565 to (319.18, 36.82, -150.09) mm, rotated rx -179.9 ry 0 rz -90 deg; joints [37.175, -66.119, 103.104, -127.665, 49.744, 140.984]
  MoveL 1566 to (317.03, 36.74, -150.44) mm, rotated rx -179.9 ry 0 rz -90 deg; joints [37.098, -66.178, 103.197, -127.766, 49.716, 141.069]
  MoveL 1567 to (315.14, 36.66, -151.54) mm, rotated rx -179.9 ry 0 rz -90 deg; joints [37.011, -66.191, 103.224, -127.863, 49.67, 141.139]
  MoveL 1568 to (313.77, 36.59, -153.24) mm, rotated rx -179.9 ry 0 rz -90 deg; joints [36.927, -66.156, 103.181, -127.944, 49.612, 141.185]
  MoveL 1569 to (313.09, 36.51, -155.32) mm, rotated rx -179.9 ry 0 rz -90 deg; joints [36.855, -66.077, 103.074, -127.998, 49.55, 141.203]
  MoveL 1570 to (313.2, 36.43, -157.5) mm, rotated rx -179.9 ry 0 rz -90 deg; joints [36.806, -65.965, 102.918, -128.019, 49.492, 141.189]
  MoveL 1571 to (314.07, 36.36, -159.5) mm, rotated rx -179.9 ry 0 rz -90 deg; joints [36.787, -65.834, 102.734, -128.003, 49.447, 141.147]
  MoveL 1572 to (315.61, 36.28, -161.06) mm, rotated rx -179.9 ry 0 rz -90 deg; joints [36.798, -65.701, 102.546, -127.954, 49.42, 141.082]
  MoveL 1573 to (317.59, 36.2, -161.97) mm, rotated rx -179.9 ry 0 rz -90 deg; joints [36.84, -65.582, 102.378, -127.879, 49.416, 141.004]
  MoveL 1574 to (319.77, 36.13, -162.11) mm, rotated rx -179.9 ry 0 rz -90 deg; joints [36.905, -65.494, 102.254, -127.787, 49.436, 140.924]
  MoveL 1575 to (321.86, 36.05, -161.46) mm, rotated rx -179.9 ry 0 rz -90 deg; joints [36.987, -65.448, 102.19, -127.693, 49.477, 140.853]
  MoveL 1576 to (323.58, 35.97, -160.12) mm, rotated rx -179.9 ry 0 rz -90 deg; joints [37.073, -65.449, 102.195, -127.607, 49.534, 140.802]
  MoveL 1577 to (324.71, 35.9, -158.25) mm, rotated rx -179.9 ry 0 rz -90 deg; joints [37.154, -65.496, 102.268, -127.543, 49.601, 140.777]
  MoveL 1578 to (325.1, 35.82, -156.1) mm, rotated rx -179.9 ry 0 rz -90 deg; joints [37.218, -65.584, 102.4, -127.508, 49.668, 140.782]
  MoveL 1579 to (324.7, 35.74, -153.95) mm, rotated rx -179.9 ry 0 rz -90 deg; joints [37.257, -65.7, 102.574, -127.508, 49.729, 140.818]
  MoveL 1580 to (323.56, 35.67, -152.09) mm, rotated rx -179.9 ry 0 rz -90 deg; joints [37.266, -65.829, 102.768, -127.542, 49.774, 140.879]
  MoveL 1581 to (321.83, 35.59, -150.75) mm, rotated rx -179.9 ry 0 rz -90 deg; joints [37.243, -65.954, 102.957, -127.607, 49.798, 140.959]
  MoveL 1582 to (319.74, 35.51, -150.12) mm, rotated rx -179.9 ry 0 rz -90 deg; joints [37.192, -66.059, 103.115, -127.696, 49.799, 141.048]
  MoveL 1583 to (317.56, 35.44, -150.28) mm, rotated rx -179.9 ry 0 rz -90 deg; joints [37.119, -66.128, 103.223, -127.796, 49.777, 141.135]
  MoveL 1584 to (315.58, 35.36, -151.2) mm, rotated rx -179.9 ry 0 rz -90 deg; joints [37.034, -66.153, 103.267, -127.895, 49.735, 141.21]
  MoveL 1585 to (314.05, 35.28, -152.77) mm, rotated rx -179.9 ry 0 rz -90 deg; joints [36.948, -66.129, 103.242, -127.981, 49.679, 141.262]
  MoveL 1586 to (313.19, 35.2, -154.77) mm, rotated rx -179.9 ry 0 rz -90 deg; joints [36.872, -66.061, 103.15, -128.043, 49.617, 141.287]
  MoveL 1587 to (313.09, 35.13, -156.96) mm, rotated rx -179.9 ry 0 rz -90 deg; joints [36.817, -65.956, 103.005, -128.073, 49.558, 141.281]
  MoveL 1588 to (313.78, 35.05, -159.03) mm, rotated rx -179.9 ry 0 rz -90 deg; joints [36.789, -65.828, 102.826, -128.066, 49.509, 141.246]
  MoveL 1589 to (315.17, 34.97, -160.72) mm, rotated rx -179.9 ry 0 rz -90 deg; joints [36.793, -65.694, 102.636, -128.025, 49.477, 141.186]
  MoveL 1590 to (317.06, 34.9, -161.81) mm, rotated rx -179.9 ry 0 rz -90 deg; joints [36.827, -65.57, 102.461, -127.955, 49.467, 141.11]
  MoveL 1591 to (319.22, 34.82, -162.15) mm, rotated rx -179.9 ry 0 rz -90 deg; joints [36.888, -65.474, 102.324, -127.867, 49.48, 141.03]
  MoveL 1592 to (321.36, 34.74, -161.7) mm, rotated rx -179.9 ry 0 rz -90 deg; joints [36.966, -65.416, 102.244, -127.772, 49.516, 140.956]
  MoveL 1593 to (323.2, 34.67, -160.52) mm, rotated rx -179.9 ry 0 rz -90 deg; joints [37.052, -65.405, 102.231, -127.683, 49.57, 140.899]
  MoveL 1594 to (324.49, 34.59, -158.76) mm, rotated rx -179.9 ry 0 rz -90 deg; joints [37.135, -65.44, 102.287, -127.612, 49.635, 140.866]
  MoveL 1595 to (325.08, 34.51, -156.65) mm, rotated rx -179.9 ry 0 rz -90 deg; joints [37.204, -65.519, 102.406, -127.569, 49.703, 140.864]
  MoveL 1596 to (324.87, 34.44, -154.48) mm, rotated rx -179.9 ry 0 rz -90 deg; joints [37.25, -65.629, 102.572, -127.56, 49.766, 140.892]
  MoveL 1597 to (323.91, 34.36, -152.52) mm, rotated rx -179.9 ry 0 rz -90 deg; joints [37.267, -65.757, 102.763, -127.586, 49.815, 140.948]
  MoveL 1598 to (322.31, 34.28, -151.03) mm, rotated rx -179.9 ry 0 rz -90 deg; joints [37.252, -65.884, 102.955, -127.644, 49.846, 141.024]
  MoveL 1599 to (320.28, 34.21, -150.21) mm, rotated rx -179.9 ry 0 rz -90 deg; joints [37.208, -65.995, 103.123, -127.727, 49.853, 141.112]
  MoveL 1600 to (318.1, 34.13, -150.16) mm, rotated rx -179.9 ry 0 rz -90 deg; joints [37.14, -66.074, 103.246, -127.825, 49.836, 141.2]
  MoveL 1601 to (316.04, 34.05, -150.9) mm, rotated rx -179.9 ry 0 rz -90 deg; joints [37.057, -66.111, 103.307, -127.926, 49.799, 141.279]
  MoveL 1602 to (314.38, 33.98, -152.32) mm, rotated rx -179.9 ry 0 rz -90 deg; joints [36.97, -66.1, 103.299, -128.017, 49.746, 141.338]
  MoveL 1603 to (313.34, 33.9, -154.24) mm, rotated rx -179.9 ry 0 rz -90 deg; joints [36.89, -66.042, 103.223, -128.086, 49.685, 141.37]
  MoveL 1604 to (313.04, 33.82, -156.4) mm, rotated rx -179.9 ry 0 rz -90 deg; joints [36.829, -65.945, 103.09, -128.124, 49.624, 141.372]
  MoveL 1605 to (313.54, 33.75, -158.53) mm, rotated rx -179.9 ry 0 rz -90 deg; joints [36.794, -65.822, 102.917, -128.127, 49.572, 141.343]
  MoveL 1606 to (314.76, 33.67, -160.34) mm, rotated rx -179.9 ry 0 rz -90 deg; joints [36.79, -65.688, 102.727, -128.094, 49.535, 141.289]
  MoveL 1607 to (316.55, 33.59, -161.6) mm, rotated rx -179.9 ry 0 rz -90 deg; joints [36.817, -65.56, 102.546, -128.031, 49.519, 141.216]
  MoveL 1608 to (318.67, 33.52, -162.14) mm, rotated rx -179.9 ry 0 rz -90 deg; joints [36.871, -65.455, 102.398, -127.946, 49.526, 141.136]
  MoveL 1609 to (320.84, 33.44, -161.88) mm, rotated rx -179.9 ry 0 rz -90 deg; joints [36.946, -65.387, 102.302, -127.851, 49.556, 141.059]
  MoveL 1610 to (322.78, 33.36, -160.88) mm, rotated rx -179.9 ry 0 rz -90 deg; joints [37.031, -65.363, 102.271, -127.759, 49.606, 140.997]
  MoveL 1611 to (324.23, 33.29, -159.24) mm, rotated rx -179.9 ry 0 rz -90 deg; joints [37.116, -65.388, 102.31, -127.683, 49.669, 140.958]
  MoveL 1612 to (325, 33.21, -157.2) mm, rotated rx -179.9 ry 0 rz -90 deg; joints [37.189, -65.456, 102.415, -127.632, 49.737, 140.948]
  MoveL 1613 to (325, 33.13, -155.02) mm, rotated rx -179.9 ry 0 rz -90 deg; joints [37.242, -65.559, 102.57, -127.614, 49.802, 140.969]
  MoveL 1614 to (324.22, 33.06, -152.98) mm, rotated rx -179.9 ry 0 rz -90 deg; joints [37.266, -65.684, 102.757, -127.631, 49.856, 141.018]
  MoveL 1615 to (322.76, 32.98, -151.35) mm, rotated rx -179.9 ry 0 rz -90 deg; joints [37.26, -65.813, 102.952, -127.682, 49.892, 141.09]
  MoveL 1616 to (320.82, 32.9, -150.34) mm, rotated rx -179.9 ry 0 rz -90 deg; joints [37.222, -65.93, 103.128, -127.759, 49.905, 141.175]
  MoveL 1617 to (318.65, 32.83, -150.1) mm, rotated rx -179.9 ry 0 rz -90 deg; joints [37.159, -66.018, 103.264, -127.855, 49.894, 141.264]
  MoveL 1618 to (316.53, 32.75, -150.64) mm, rotated rx -179.9 ry 0 rz -90 deg; joints [37.079, -66.066, 103.342, -127.956, 49.862, 141.346]
  MoveL 1619 to (314.75, 32.67, -151.91) mm, rotated rx -179.9 ry 0 rz -90 deg; joints [36.992, -66.067, 103.351, -128.051, 49.813, 141.411]
  MoveL 1620 to (313.53, 32.6, -153.72) mm, rotated rx -179.9 ry 0 rz -90 deg; joints [36.91, -66.021, 103.292, -128.126, 49.753, 141.451]
  MoveL 1621 to (313.04, 32.52, -155.85) mm, rotated rx -179.9 ry 0 rz -90 deg; joints [36.843, -65.933, 103.172, -128.173, 49.691, 141.46]
  MoveL 1622 to (313.34, 32.44, -158.01) mm, rotated rx -179.9 ry 0 rz -90 deg; joints [36.801, -65.815, 103.007, -128.185, 49.636, 141.439]
  MoveL 1623 to (314.39, 32.37, -159.93) mm, rotated rx -179.9 ry 0 rz -90 deg; joints [36.788, -65.682, 102.819, -128.161, 49.594, 141.391]
  MoveL 1624 to (316.06, 32.29, -161.34) mm, rotated rx -179.9 ry 0 rz -90 deg; joints [36.808, -65.551, 102.634, -128.104, 49.573, 141.322]
  MoveL 1625 to (318.12, 32.21, -162.07) mm, rotated rx -179.9 ry 0 rz -90 deg; joints [36.856, -65.439, 102.475, -128.024, 49.574, 141.242]
  MoveL 1626 to (320.3, 32.14, -162.02) mm, rotated rx -179.9 ry 0 rz -90 deg; joints [36.926, -65.361, 102.364, -127.93, 49.598, 141.163]
  MoveL 1627 to (322.32, 32.06, -161.2) mm, rotated rx -179.9 ry 0 rz -90 deg; joints [37.01, -65.325, 102.316, -127.837, 49.643, 141.097]
  MoveL 1628 to (323.92, 31.98, -159.7) mm, rotated rx -179.9 ry 0 rz -90 deg; joints [37.096, -65.338, 102.338, -127.755, 49.704, 141.051]
  MoveL 1629 to (324.88, 31.91, -157.74) mm, rotated rx -179.9 ry 0 rz -90 deg; joints [37.173, -65.395, 102.426, -127.697, 49.771, 141.034]
  MoveL 1630 to (325.08, 31.83, -155.56) mm, rotated rx -179.9 ry 0 rz -90 deg; joints [37.232, -65.491, 102.571, -127.671, 49.838, 141.047]
  MoveL 1631 to (324.48, 31.75, -153.46) mm, rotated rx -179.9 ry 0 rz -90 deg; joints [37.264, -65.612, 102.752, -127.679, 49.895, 141.089]
  MoveL 1632 to (323.18, 31.68, -151.71) mm, rotated rx -179.9 ry 0 rz -90 deg; joints [37.265, -65.741, 102.947, -127.721, 49.936, 141.156]
  MoveL 1633 to (321.34, 31.6, -150.53) mm, rotated rx -179.9 ry 0 rz -90 deg; joints [37.235, -65.863, 103.13, -127.792, 49.955, 141.239]
  MoveL 1634 to (319.2, 31.52, -150.09) mm, rotated rx -179.9 ry 0 rz -90 deg; joints [37.178, -65.959, 103.278, -127.884, 49.951, 141.328]
  MoveL 1635 to (317.04, 31.45, -150.43) mm, rotated rx -179.9 ry 0 rz -90 deg; joints [37.101, -66.018, 103.372, -127.986, 49.924, 141.413]
  MoveL 1636 to (315.15, 31.37, -151.53) mm, rotated rx -179.9 ry 0 rz -90 deg; joints [37.015, -66.031, 103.399, -128.083, 49.878, 141.483]
  MoveL 1637 to (313.78, 31.29, -153.22) mm, rotated rx -179.9 ry 0 rz -90 deg; joints [36.93, -65.997, 103.357, -128.164, 49.821, 141.529]
  MoveL 1638 to (313.09, 31.22, -155.3) mm, rotated rx -179.9 ry 0 rz -90 deg; joints [36.858, -65.918, 103.251, -128.219, 49.759, 141.546]
  MoveL 1639 to (313.19, 31.14, -157.48) mm, rotated rx -179.9 ry 0 rz -90 deg; joints [36.809, -65.807, 103.095, -128.24, 49.701, 141.533]
  MoveL 1640 to (314.06, 31.06, -159.48) mm, rotated rx -179.9 ry 0 rz -90 deg; joints [36.789, -65.676, 102.911, -128.225, 49.655, 141.491]
  MoveL 1641 to (315.59, 30.99, -161.05) mm, rotated rx -179.9 ry 0 rz -90 deg; joints [36.801, -65.543, 102.722, -128.176, 49.628, 141.426]
  MoveL 1642 to (317.57, 30.91, -161.96) mm, rotated rx -179.9 ry 0 rz -90 deg; joints [36.842, -65.425, 102.555, -128.101, 49.623, 141.348]
  MoveL 1643 to (319.75, 30.83, -162.11) mm, rotated rx -179.9 ry 0 rz -90 deg; joints [36.907, -65.337, 102.43, -128.01, 49.642, 141.268]
  MoveL 1644 to (321.84, 30.76, -161.47) mm, rotated rx -179.9 ry 0 rz -90 deg; joints [36.989, -65.29, 102.365, -127.915, 49.682, 141.198]
  MoveL 1645 to (323.57, 30.68, -160.13) mm, rotated rx -179.9 ry 0 rz -90 deg; joints [37.075, -65.29, 102.369, -127.829, 49.739, 141.146]
  MoveL 1646 to (324.7, 30.6, -158.27) mm, rotated rx -179.9 ry 0 rz -90 deg; joints [37.156, -65.337, 102.442, -127.764, 49.805, 141.121]
  MoveL 1647 to (325.1, 30.52, -156.12) mm, rotated rx -179.9 ry 0 rz -90 deg; joints [37.22, -65.424, 102.574, -127.729, 49.873, 141.126]
  MoveL 1648 to (325.1, 30.52, -1) mm, rotated rx -179.9 ry 0 rz -90 deg; joints [41.29, -72.681, 112.645, -125.473, 54.106, 141.584]
  MoveL 1649 to (-325.1, 30.53, -1) mm, rotated rx -179.9 ry 0 rz -90 deg; joints [12.691, -91.861, 135.095, -161.5, 43.795, 166.844]
  MoveL 1650 to (-325.1, 30.53, -311.23) mm, rotated rx -179.9 ry 0 rz -90 deg; joints [9.718, -72.497, 112.988, -164.952, 40.531, 168.823]
  MoveL 1651 to (325.1, 30.53, -311.23) mm, rotated rx -179.9 ry 0 rz -90 deg; joints [33.789, -57.633, 90.789, -128.413, 45.202, 139.212]
  MoveL 1652 to (325.1, 30.52, -156.12) mm, rotated rx -179.9 ry 0 rz -90 deg; joints [37.22, -65.424, 102.574, -127.729, 49.873, 141.126]
  MoveC 1653 to (323.81, 30.53, -151.87) mm, rotated rx -179.9 ry 0 rz -90 deg; joints [37.282, -65.676, 102.94, -127.743, 49.982, 141.205] to (320.39, 30.52, -149.05) mm, rotated rx -179.9 ry 0 rz -90 deg; joints [37.241, -65.936, 103.32, -127.863, 50.03, 141.355]
  MoveL 1654 to (320.39, 30.53, -149.05) mm, rotated rx -179.9 ry 0 rz -90 deg; joints [37.241, -65.936, 103.32, -127.863, 50.03, 141.355]
  MoveC 1655 to (316.96, 30.53, -146.23) mm, rotated rx -179.9 ry 0 rz -90 deg; joints [37.201, -66.196, 103.698, -127.983, 50.078, 141.502] to (315.68, 30.53, -141.98) mm, rotated rx -179.9 ry 0 rz -90 deg; joints [37.263, -66.447, 104.06, -127.993, 50.185, 141.577]
  MoveL 1656 to (315.68, 30.52, -141.98) mm, rotated rx -179.9 ry 0 rz -90 deg; joints [37.263, -66.447, 104.06, -127.993, 50.185, 141.577]
  MoveL 1657 to (315.68, 30.53, -14.28) mm, rotated rx -179.9 ry 0 rz -90 deg; joints [40.606, -72.444, 112.344, -126.098, 53.643, 141.9]
  MoveC 1658 to (314.55, 30.53, -11.55) mm, rotated rx -179.9 ry 0 rz -90 deg; joints [40.646, -72.613, 112.569, -126.093, 53.701, 141.934] to (311.82, 30.52, -10.43) mm, rotated rx -179.9 ry 0 rz -90 deg; joints [40.588, -72.77, 112.782, -126.181, 53.698, 142.021]
  MoveL 1659 to (311.82, 30.52, -10.43) mm, rotated rx -179.9 ry 0 rz -90 deg; joints [40.588, -72.77, 112.782, -126.181, 53.698, 142.021]
  MoveL 1660 to (-311.82, 30.52, -10.43) mm, rotated rx -179.9 ry 0 rz -90 deg; joints [13.295, -91.021, 134.29, -160.665, 43.97, 166.26]
  MoveC 1661 to (-314.55, 30.52, -11.55) mm, rotated rx -179.9 ry 0 rz -90 deg; joints [13.133, -90.988, 134.259, -160.893, 43.935, 166.422] to (-315.68, 30.52, -14.28) mm, rotated rx -179.9 ry 0 rz -90 deg; joints [13.037, -90.823, 134.101, -161.029, 43.919, 166.52]
  MoveL 1662 to (-315.68, 30.52, -14.28) mm, rotated rx -179.9 ry 0 rz -90 deg; joints [13.037, -90.823, 134.101, -161.029, 43.919, 166.52]
  MoveL 1663 to (-315.68, 30.52, -297.96) mm, rotated rx -179.9 ry 0 rz -90 deg; joints [10.223, -73.187, 113.9, -164.263, 40.846, 168.347]
  MoveC 1664 to (-314.55, 30.52, -300.68) mm, rotated rx -179.9 ry 0 rz -90 deg; joints [10.25, -73.013, 113.67, -164.204, 40.797, 168.293] to (-311.82, 30.53, -301.81) mm, rotated rx -179.9 ry 0 rz -90 deg; joints [10.357, -72.918, 113.541, -164.033, 40.788, 168.159]
  MoveL 1665 to (-311.82, 30.53, -301.81) mm, rotated rx -179.9 ry 0 rz -90 deg; joints [10.357, -72.918, 113.541, -164.033, 40.788, 168.159]
  MoveL 1666 to (311.82, 30.52, -301.81) mm, rotated rx -179.9 ry 0 rz -90 deg; joints [33.576, -58.587, 92.296, -129.066, 45.41, 139.975]
  MoveC 1667 to (314.55, 30.52, -300.68) mm, rotated rx -179.9 ry 0 rz -90 deg; joints [33.683, -58.552, 92.238, -128.935, 45.465, 139.872] to (315.68, 30.52, -297.96) mm, rotated rx -179.9 ry 0 rz -90 deg; joints [33.773, -58.655, 92.398, -128.881, 45.558, 139.867]
  MoveL 1668 to (315.68, 30.52, -297.96) mm, rotated rx -179.9 ry 0 rz -90 deg; joints [33.773, -58.655, 92.398, -128.881, 45.558, 139.867]
  MoveL 1669 to (315.68, 30.52, -141.98) mm, rotated rx -179.9 ry 0 rz -90 deg; joints [37.263, -66.447, 104.06, -127.993, 50.185, 141.577]
  MoveC 1670 to (314.4, 30.52, -137.76) mm, rotated rx -179.9 ry 0 rz -90 deg; joints [37.325, -66.696, 104.419, -128.001, 50.291, 141.65] to (311, 30.53, -134.96) mm, rotated rx -179.9 ry 0 rz -90 deg; joints [37.285, -66.954, 104.791, -128.117, 50.336, 141.792]
  MoveL 1671 to (311, 30.53, -134.96) mm, rotated rx -179.9 ry 0 rz -90 deg; joints [37.285, -66.954, 104.791, -128.117, 50.336, 141.792]
  MoveC 1672 to (307.59, 30.52, -132.16) mm, rotated rx -179.9 ry 0 rz -90 deg; joints [37.244, -67.212, 105.162, -128.232, 50.381, 141.934] to (306.32, 30.52, -127.94) mm, rotated rx -179.9 ry 0 rz -90 deg; joints [37.307, -67.461, 105.517, -128.237, 50.486, 142.002]
  MoveL 1673 to (306.32, 30.52, -127.94) mm, rotated rx -179.9 ry 0 rz -90 deg; joints [37.307, -67.461, 105.517, -128.237, 50.486, 142.002]
  MoveL 1674 to (306.32, 30.53, -23.64) mm, rotated rx -179.9 ry 0 rz -90 deg; joints [40.037, -72.374, 112.264, -126.649, 53.286, 142.212]
  MoveC 1675 to (305.19, 30.53, -20.92) mm, rotated rx -179.9 ry 0 rz -90 deg; joints [40.076, -72.543, 112.491, -126.645, 53.343, 142.247] to (302.46, 30.53, -19.79) mm, rotated rx -179.9 ry 0 rz -90 deg; joints [40.017, -72.7, 112.702, -126.735, 53.34, 142.335]
  MoveL 1676 to (302.46, 30.53, -19.79) mm, rotated rx -179.9 ry 0 rz -90 deg; joints [40.017, -72.7, 112.702, -126.735, 53.34, 142.335]
  MoveL 1677 to (-302.46, 30.52, -19.79) mm, rotated rx -179.9 ry 0 rz -90 deg; joints [13.676, -90.249, 133.537, -160.14, 44.083, 165.894]
  MoveC 1678 to (-305.19, 30.52, -20.92) mm, rotated rx -179.9 ry 0 rz -90 deg; joints [13.516, -90.217, 133.508, -160.364, 44.046, 166.053] to (-306.32, 30.52, -23.64) mm, rotated rx -179.9 ry 0 rz -90 deg; joints [13.421, -90.054, 133.349, -160.499, 44.027, 166.149]
  MoveL 1679 to (-306.32, 30.53, -23.64) mm, rotated rx -179.9 ry 0 rz -90 deg; joints [13.421, -90.054, 133.349, -160.499, 44.027, 166.149]
  MoveL 1680 to (-306.32, 30.52, -288.59) mm, rotated rx -179.9 ry 0 rz -90 deg; joints [10.701, -73.641, 114.493, -163.594, 41.08, 167.875]
  MoveC 1681 to (-305.19, 30.53, -291.32) mm, rotated rx -179.9 ry 0 rz -90 deg; joints [10.727, -73.467, 114.263, -163.537, 41.032, 167.822] to (-302.46, 30.52, -292.45) mm, rotated rx -179.9 ry 0 rz -90 deg; joints [10.835, -73.37, 114.134, -163.366, 41.025, 167.689]
  MoveL 1682 to (-302.46, 30.52, -292.45) mm, rotated rx -179.9 ry 0 rz -90 deg; joints [10.835, -73.37, 114.134, -163.366, 41.025, 167.689]
  MoveL 1683 to (302.46, 30.53, -292.45) mm, rotated rx -179.9 ry 0 rz -90 deg; joints [33.48, -59.396, 93.562, -129.517, 45.637, 140.541]
  MoveC 1684 to (305.19, 30.52, -291.32) mm, rotated rx -179.9 ry 0 rz -90 deg; joints [33.587, -59.362, 93.506, -129.385, 45.692, 140.439] to (306.32, 30.52, -288.59) mm, rotated rx -179.9 ry 0 rz -90 deg; joints [33.678, -59.465, 93.663, -129.329, 45.785, 140.431]
  MoveL 1685 to (306.32, 30.52, -288.59) mm, rotated rx -179.9 ry 0 rz -90 deg; joints [33.678, -59.465, 93.663, -129.329, 45.785, 140.431]
  MoveL 1686 to (306.32, 30.52, -127.94) mm, rotated rx -179.9 ry 0 rz -90 deg; joints [37.307, -67.461, 105.517, -128.237, 50.486, 142.002]
  MoveC 1687 to (305.04, 30.52, -123.72) mm, rotated rx -179.9 ry 0 rz -90 deg; joints [37.37, -67.709, 105.871, -128.24, 50.589, 142.069] to (301.63, 30.53, -120.92) mm, rotated rx -179.9 ry 0 rz -90 deg; joints [37.329, -67.967, 106.238, -128.353, 50.632, 142.206]
  MoveL 1688 to (301.63, 30.52, -120.92) mm, rotated rx -179.9 ry 0 rz -90 deg; joints [37.329, -67.967, 106.238, -128.353, 50.632, 142.206]
  MoveC 1689 to (298.23, 30.53, -118.11) mm, rotated rx -179.9 ry 0 rz -90 deg; joints [37.288, -68.224, 106.604, -128.465, 50.675, 142.342] to (296.95, 30.52, -113.9) mm, rotated rx -179.9 ry 0 rz -90 deg; joints [37.351, -68.473, 106.954, -128.465, 50.777, 142.405]
  MoveL 1690 to (296.95, 30.53, -113.9) mm, rotated rx -179.9 ry 0 rz -90 deg; joints [37.351, -68.473, 106.954, -128.465, 50.777, 142.405]
  MoveL 1691 to (296.95, 30.53, -33) mm, rotated rx -179.9 ry 0 rz -90 deg; joints [39.469, -72.296, 112.174, -127.202, 52.93, 142.526]
  MoveC 1692 to (295.82, 30.52, -30.28) mm, rotated rx -179.9 ry 0 rz -90 deg; joints [39.507, -72.466, 112.401, -127.199, 52.987, 142.562] to (293.1, 30.53, -29.15) mm, rotated rx -179.9 ry 0 rz -90 deg; joints [39.447, -72.623, 112.612, -127.291, 52.984, 142.651]
  MoveL 1693 to (293.1, 30.52, -29.15) mm, rotated rx -179.9 ry 0 rz -90 deg; joints [39.447, -72.623, 112.612, -127.291, 52.984, 142.651]
  MoveL 1694 to (-293.1, 30.53, -29.15) mm, rotated rx -179.9 ry 0 rz -90 deg; joints [14.049, -89.48, 132.776, -159.624, 44.183, 165.531]
  MoveC 1695 to (-295.82, 30.53, -30.28) mm, rotated rx -179.9 ry 0 rz -90 deg; joints [13.891, -89.45, 132.748, -159.845, 44.145, 165.688] to (-296.95, 30.53, -33) mm, rotated rx -179.9 ry 0 rz -90 deg; joints [13.796, -89.289, 132.589, -159.978, 44.123, 165.782]
  MoveL 1696 to (-296.95, 30.52, -33) mm, rotated rx -179.9 ry 0 rz -90 deg; joints [13.796, -89.289, 132.589, -159.978, 44.123, 165.782]
  MoveL 1697 to (-296.95, 30.52, -279.23) mm, rotated rx -179.9 ry 0 rz -90 deg; joints [11.184, -74.09, 115.075, -162.921, 41.313, 167.402]
  MoveC 1698 to (-295.82, 30.53, -281.95) mm, rotated rx -179.9 ry 0 rz -90 deg; joints [11.21, -73.915, 114.847, -162.866, 41.267, 167.35] to (-293.1, 30.53, -283.08) mm, rotated rx -179.9 ry 0 rz -90 deg; joints [11.318, -73.817, 114.716, -162.696, 41.26, 167.218]
  MoveL 1699 to (-293.1, 30.52, -283.08) mm, rotated rx -179.9 ry 0 rz -90 deg; joints [11.318, -73.817, 114.716, -162.696, 41.26, 167.218]
  MoveL 1700 to (293.1, 30.53, -283.08) mm, rotated rx -179.9 ry 0 rz -90 deg; joints [33.381, -60.201, 94.811, -129.956, 45.859, 141.091]
  MoveC 1701 to (295.82, 30.53, -281.95) mm, rotated rx -179.9 ry 0 rz -90 deg; joints [33.49, -60.167, 94.755, -129.823, 45.914, 140.988] to (296.95, 30.53, -279.23) mm, rotated rx -179.9 ry 0 rz -90 deg; joints [33.581, -60.269, 94.911, -129.764, 46.006, 140.978]
  MoveL 1702 to (296.95, 30.52, -279.23) mm, rotated rx -179.9 ry 0 rz -90 deg; joints [33.581, -60.269, 94.911, -129.764, 46.006, 140.978]
  MoveL 1703 to (296.95, 30.53, -113.9) mm, rotated rx -179.9 ry 0 rz -90 deg; joints [37.351, -68.473, 106.954, -128.465, 50.777, 142.405]
  MoveC 1704 to (295.67, 30.52, -109.68) mm, rotated rx -179.9 ry 0 rz -90 deg; joints [37.415, -68.721, 107.303, -128.463, 50.878, 142.466] to (292.27, 30.52, -106.87) mm, rotated rx -179.9 ry 0 rz -90 deg; joints [37.374, -68.979, 107.666, -128.572, 50.919, 142.598]
  MoveL 1705 to (292.27, 30.52, -106.87) mm, rotated rx -179.9 ry 0 rz -90 deg; joints [37.374, -68.979, 107.666, -128.572, 50.919, 142.598]
  MoveC 1706 to (288.87, 30.52, -104.07) mm, rotated rx -179.9 ry 0 rz -90 deg; joints [37.333, -69.236, 108.027, -128.681, 50.959, 142.729] to (287.59, 30.53, -99.85) mm, rotated rx -179.9 ry 0 rz -90 deg; joints [37.397, -69.484, 108.372, -128.676, 51.058, 142.786]
  MoveL 1707 to (287.59, 30.53, -99.85) mm, rotated rx -179.9 ry 0 rz -90 deg; joints [37.397, -69.484, 108.372, -128.676, 51.058, 142.786]
  MoveL 1708 to (287.59, 30.52, -42.37) mm, rotated rx -179.9 ry 0 rz -90 deg; joints [38.902, -72.211, 112.073, -127.757, 52.575, 142.843]
  MoveC 1709 to (286.46, 30.52, -39.64) mm, rotated rx -179.9 ry 0 rz -90 deg; joints [38.938, -72.382, 112.301, -127.756, 52.632, 142.879] to (283.74, 30.52, -38.51) mm, rotated rx -179.9 ry 0 rz -90 deg; joints [38.878, -72.537, 112.511, -127.849, 52.629, 142.97]
  MoveL 1710 to (283.74, 30.53, -38.51) mm, rotated rx -179.9 ry 0 rz -90 deg; joints [38.878, -72.537, 112.511, -127.849, 52.629, 142.97]
  MoveL 1711 to (-283.74, 30.53, -38.51) mm, rotated rx -179.9 ry 0 rz -90 deg; joints [14.414, -88.715, 132.006, -159.116, 44.272, 165.172]
  MoveC 1712 to (-286.46, 30.53, -39.64) mm, rotated rx -179.9 ry 0 rz -90 deg; joints [14.257, -88.686, 131.979, -159.334, 44.233, 165.326] to (-287.59, 30.53, -42.37) mm, rotated rx -179.9 ry 0 rz -90 deg; joints [14.163, -88.528, 131.819, -159.465, 44.208, 165.418]
  MoveL 1713 to (-287.59, 30.53, -42.37) mm, rotated rx -179.9 ry 0 rz -90 deg; joints [14.163, -88.528, 131.819, -159.465, 44.208, 165.418]
  MoveL 1714 to (-287.59, 30.52, -269.87) mm, rotated rx -179.9 ry 0 rz -90 deg; joints [11.674, -74.534, 115.647, -162.245, 41.545, 166.928]
  MoveC 1715 to (-286.46, 30.52, -272.59) mm, rotated rx -179.9 ry 0 rz -90 deg; joints [11.698, -74.359, 115.42, -162.191, 41.501, 166.877] to (-283.74, 30.52, -273.72) mm, rotated rx -179.9 ry 0 rz -90 deg; joints [11.806, -74.259, 115.288, -162.021, 41.496, 166.746]
  MoveL 1716 to (-283.74, 30.52, -273.72) mm, rotated rx -179.9 ry 0 rz -90 deg; joints [11.806, -74.259, 115.288, -162.021, 41.496, 166.746]
  MoveL 1717 to (283.74, 30.52, -273.72) mm, rotated rx -179.9 ry 0 rz -90 deg; joints [33.281, -61, 96.043, -130.384, 46.075, 141.624]
  MoveC 1718 to (286.46, 30.53, -272.59) mm, rotated rx -179.9 ry 0 rz -90 deg; joints [33.391, -60.967, 95.989, -130.25, 46.13, 141.522] to (287.59, 30.52, -269.87) mm, rotated rx -179.9 ry 0 rz -90 deg; joints [33.483, -61.069, 96.143, -130.189, 46.221, 141.509]
  MoveL 1719 to (287.59, 30.53, -269.87) mm, rotated rx -179.9 ry 0 rz -90 deg; joints [33.483, -61.069, 96.143, -130.189, 46.221, 141.509]
  MoveL 1720 to (287.59, 30.53, -99.85) mm, rotated rx -179.9 ry 0 rz -90 deg; joints [37.397, -69.484, 108.372, -128.676, 51.058, 142.786]
  MoveC 1721 to (286.31, 30.53, -95.63) mm, rotated rx -179.9 ry 0 rz -90 deg; joints [37.462, -69.733, 108.716, -128.67, 51.158, 142.841] to (282.91, 30.53, -92.83) mm, rotated rx -179.9 ry 0 rz -90 deg; joints [37.421, -69.99, 109.075, -128.776, 51.196, 142.968]
  MoveL 1722 to (282.91, 30.52, -92.83) mm, rotated rx -179.9 ry 0 rz -90 deg; joints [37.421, -69.99, 109.075, -128.776, 51.196, 142.968]
  MoveC 1723 to (279.5, 30.52, -90.03) mm, rotated rx -179.9 ry 0 rz -90 deg; joints [37.379, -70.247, 109.432, -128.881, 51.233, 143.094] to (278.23, 30.52, -85.81) mm, rotated rx -179.9 ry 0 rz -90 deg; joints [37.445, -70.496, 109.772, -128.872, 51.33, 143.145]
  MoveL 1724 to (278.23, 30.52, -85.81) mm, rotated rx -179.9 ry 0 rz -90 deg; joints [37.445, -70.496, 109.772, -128.872, 51.33, 143.145]
  MoveL 1725 to (278.23, 30.52, -51.73) mm, rotated rx -179.9 ry 0 rz -90 deg; joints [38.337, -72.118, 111.961, -128.314, 52.221, 143.162]
  MoveC 1726 to (277.1, 30.53, -49.01) mm, rotated rx -179.9 ry 0 rz -90 deg; joints [38.371, -72.289, 112.19, -128.315, 52.278, 143.199] to (274.37, 30.52, -47.88) mm, rotated rx -179.9 ry 0 rz -90 deg; joints [38.31, -72.443, 112.399, -128.41, 52.275, 143.29]
  MoveL 1727 to (274.37, 30.52, -47.88) mm, rotated rx -179.9 ry 0 rz -90 deg; joints [38.31, -72.443, 112.399, -128.41, 52.275, 143.29]
  MoveL 1728 to (-274.37, 30.53, -47.88) mm, rotated rx -179.9 ry 0 rz -90 deg; joints [14.772, -87.954, 131.227, -158.616, 44.35, 164.815]
  MoveC 1729 to (-277.1, 30.53, -49.01) mm, rotated rx -179.9 ry 0 rz -90 deg; joints [14.616, -87.926, 131.201, -158.831, 44.31, 164.967] to (-278.23, 30.52, -51.73) mm, rotated rx -179.9 ry 0 rz -90 deg; joints [14.522, -87.77, 131.041, -158.961, 44.282, 165.057]
  MoveL 1730 to (-278.23, 30.52, -51.73) mm, rotated rx -179.9 ry 0 rz -90 deg; joints [14.522, -87.77, 131.041, -158.961, 44.282, 165.057]
  MoveL 1731 to (-278.23, 30.52, -260.51) mm, rotated rx -179.9 ry 0 rz -90 deg; joints [12.168, -74.973, 116.209, -161.564, 41.778, 166.453]
  MoveC 1732 to (-277.1, 30.53, -263.23) mm, rotated rx -179.9 ry 0 rz -90 deg; joints [12.192, -74.798, 115.982, -161.512, 41.735, 166.403] to (-274.37, 30.52, -264.36) mm, rotated rx -179.9 ry 0 rz -90 deg; joints [12.3, -74.696, 115.85, -161.343, 41.731, 166.273]
  MoveL 1733 to (-274.37, 30.52, -264.36) mm, rotated rx -179.9 ry 0 rz -90 deg; joints [12.3, -74.696, 115.85, -161.343, 41.731, 166.273]
  MoveL 1734 to (274.37, 30.52, -264.36) mm, rotated rx -179.9 ry 0 rz -90 deg; joints [33.18, -61.796, 97.259, -130.801, 46.286, 142.142]
  MoveC 1735 to (277.1, 30.52, -263.23) mm, rotated rx -179.9 ry 0 rz -90 deg; joints [33.29, -61.763, 97.206, -130.667, 46.341, 142.04] to (278.23, 30.52, -260.51) mm, rotated rx -179.9 ry 0 rz -90 deg; joints [33.383, -61.865, 97.359, -130.602, 46.431, 142.025]
  MoveL 1736 to (278.23, 30.52, -260.51) mm, rotated rx -179.9 ry 0 rz -90 deg; joints [33.383, -61.865, 97.359, -130.602, 46.431, 142.025]
  MoveL 1737 to (278.23, 30.52, -85.81) mm, rotated rx -179.9 ry 0 rz -90 deg; joints [37.445, -70.496, 109.772, -128.872, 51.33, 143.145]
  MoveC 1738 to (276.95, 30.52, -81.59) mm, rotated rx -179.9 ry 0 rz -90 deg; joints [37.51, -70.744, 110.112, -128.861, 51.427, 143.195] to (273.55, 30.53, -78.79) mm, rotated rx -179.9 ry 0 rz -90 deg; joints [37.469, -71.001, 110.466, -128.964, 51.463, 143.317]
  MoveL 1739 to (273.55, 30.52, -78.79) mm, rotated rx -179.9 ry 0 rz -90 deg; joints [37.469, -71.001, 110.466, -128.964, 51.463, 143.317]
  MoveC 1740 to (270.14, 30.52, -75.98) mm, rotated rx -179.9 ry 0 rz -90 deg; joints [37.426, -71.259, 110.818, -129.066, 51.497, 143.438] to (268.86, 30.53, -71.76) mm, rotated rx -179.9 ry 0 rz -90 deg; joints [37.493, -71.507, 111.155, -129.052, 51.592, 143.484]
  MoveL 1741 to (268.86, 30.53, -71.76) mm, rotated rx -179.9 ry 0 rz -90 deg; joints [37.493, -71.507, 111.155, -129.052, 51.592, 143.484]
  MoveL 1742 to (268.86, 30.53, -61.09) mm, rotated rx -179.9 ry 0 rz -90 deg; joints [37.772, -72.017, 111.839, -128.874, 51.869, 143.484]
  MoveC 1743 to (267.74, 30.52, -58.37) mm, rotated rx -179.9 ry 0 rz -90 deg; joints [37.806, -72.189, 112.069, -128.875, 51.926, 143.521] to (265.01, 30.53, -57.24) mm, rotated rx -179.9 ry 0 rz -90 deg; joints [37.743, -72.342, 112.277, -128.972, 51.922, 143.614]
  MoveL 1744 to (265.01, 30.53, -57.24) mm, rotated rx -179.9 ry 0 rz -90 deg; joints [37.743, -72.342, 112.277, -128.972, 51.922, 143.614]
  MoveL 1745 to (-265.01, 30.53, -57.24) mm, rotated rx -179.9 ry 0 rz -90 deg; joints [15.122, -87.196, 130.44, -158.123, 44.416, 164.461]
  MoveC 1746 to (-267.74, 30.53, -58.37) mm, rotated rx -179.9 ry 0 rz -90 deg; joints [14.968, -87.17, 130.415, -158.335, 44.375, 164.61] to (-268.86, 30.53, -61.09) mm, rotated rx -179.9 ry 0 rz -90 deg; joints [14.874, -87.015, 130.254, -158.463, 44.345, 164.699]
  MoveL 1747 to (-268.86, 30.52, -61.09) mm, rotated rx -179.9 ry 0 rz -90 deg; joints [14.874, -87.015, 130.254, -158.463, 44.345, 164.699]
  MoveL 1748 to (-268.86, 30.52, -251.14) mm, rotated rx -179.9 ry 0 rz -90 deg; joints [12.669, -75.407, 116.761, -160.879, 42.01, 165.977]
  MoveC 1749 to (-267.74, 30.52, -253.87) mm, rotated rx -179.9 ry 0 rz -90 deg; joints [12.691, -75.231, 116.534, -160.828, 41.968, 165.928] to (-265.01, 30.52, -255) mm, rotated rx -179.9 ry 0 rz -90 deg; joints [12.799, -75.128, 116.401, -160.661, 41.966, 165.799]
  MoveL 1750 to (-265.01, 30.53, -255) mm, rotated rx -179.9 ry 0 rz -90 deg; joints [12.799, -75.128, 116.401, -160.661, 41.966, 165.799]
  MoveL 1751 to (265.01, 30.52, -255) mm, rotated rx -179.9 ry 0 rz -90 deg; joints [33.076, -62.587, 98.46, -131.208, 46.491, 142.644]
  MoveC 1752 to (267.74, 30.53, -253.87) mm, rotated rx -179.9 ry 0 rz -90 deg; joints [33.188, -62.555, 98.408, -131.073, 46.546, 142.542] to (268.86, 30.53, -251.14) mm, rotated rx -179.9 ry 0 rz -90 deg; joints [33.281, -62.657, 98.559, -131.006, 46.636, 142.525]
  MoveL 1753 to (268.86, 30.52, -251.14) mm, rotated rx -179.9 ry 0 rz -90 deg; joints [33.281, -62.657, 98.559, -131.006, 46.636, 142.525]
  MoveL 1754 to (268.86, 30.53, -71.76) mm, rotated rx -179.9 ry 0 rz -90 deg; joints [37.493, -71.507, 111.155, -129.052, 51.592, 143.484]
  MoveC 1755 to (266.09, 30.53, -66.2) mm, rotated rx -179.9 ry 0 rz -90 deg; joints [37.544, -71.874, 111.651, -129.079, 51.704, 143.58] to (259.98, 30.52, -65.06) mm, rotated rx -179.9 ry 0 rz -90 deg; joints [37.366, -72.151, 112.028, -129.323, 51.662, 143.789]
  MoveL 1756 to (259.98, 30.53, -65.06) mm, rotated rx -179.9 ry 0 rz -90 deg; joints [37.366, -72.151, 112.028, -129.323, 51.662, 143.789]
  MoveC 1757 to (254.53, 30.52, -66.22) mm, rotated rx -179.9 ry 0 rz -90 deg; joints [37.149, -72.292, 112.224, -129.579, 51.568, 143.977] to (248.97, 30.52, -66.6) mm, rotated rx -179.9 ry 0 rz -90 deg; joints [36.948, -72.474, 112.472, -129.827, 51.492, 144.169]
  MoveL 1758 to (248.97, 30.52, -66.6) mm, rotated rx -179.9 ry 0 rz -90 deg; joints [36.948, -72.474, 112.472, -129.827, 51.492, 144.169]
  MoveL 1759 to (-255.65, 30.52, -66.6) mm, rotated rx -179.9 ry 0 rz -90 deg; joints [15.465, -86.441, 129.644, -157.637, 44.472, 164.109]
  MoveC 1760 to (-258.37, 30.53, -67.73) mm, rotated rx -179.9 ry 0 rz -90 deg; joints [15.312, -86.416, 129.619, -157.846, 44.43, 164.256] to (-259.5, 30.52, -70.46) mm, rotated rx -179.9 ry 0 rz -90 deg; joints [15.218, -86.263, 129.459, -157.972, 44.397, 164.342]
  MoveL 1761 to (-259.5, 30.53, -70.46) mm, rotated rx -179.9 ry 0 rz -90 deg; joints [15.218, -86.263, 129.459, -157.972, 44.397, 164.342]
  MoveL 1762 to (-259.5, 30.53, -241.78) mm, rotated rx -179.9 ry 0 rz -90 deg; joints [13.174, -75.836, 117.302, -160.19, 42.242, 165.499]
  MoveC 1763 to (-258.37, 30.52, -244.5) mm, rotated rx -179.9 ry 0 rz -90 deg; joints [13.196, -75.659, 117.076, -160.141, 42.202, 165.452] to (-255.65, 30.53, -245.63) mm, rotated rx -179.9 ry 0 rz -90 deg; joints [13.303, -75.555, 116.942, -159.975, 42.201, 165.324]
  MoveL 1764 to (-255.65, 30.52, -245.63) mm, rotated rx -179.9 ry 0 rz -90 deg; joints [13.303, -75.555, 116.942, -159.975, 42.201, 165.324]
  MoveL 1765 to (255.65, 30.53, -245.63) mm, rotated rx -179.9 ry 0 rz -90 deg; joints [32.971, -63.376, 99.646, -131.605, 46.69, 143.132]
  MoveC 1766 to (258.37, 30.53, -244.5) mm, rotated rx -179.9 ry 0 rz -90 deg; joints [33.083, -63.344, 99.595, -131.469, 46.745, 143.031] to (259.5, 30.52, -241.78) mm, rotated rx -179.9 ry 0 rz -90 deg; joints [33.178, -63.445, 99.745, -131.4, 46.834, 143.011]
  MoveL 1767 to (259.5, 30.52, -241.78) mm, rotated rx -179.9 ry 0 rz -90 deg; joints [33.178, -63.445, 99.745, -131.4, 46.834, 143.011]
  MoveL 1768 to (259.5, 30.52, -70.46) mm, rotated rx -179.9 ry 0 rz -90 deg; joints [37.209, -71.909, 111.706, -129.435, 51.518, 143.808]
  MoveC 1769 to (258.37, 30.52, -67.73) mm, rotated rx -179.9 ry 0 rz -90 deg; joints [37.241, -72.081, 111.937, -129.438, 51.575, 143.846] to (255.65, 30.53, -66.6) mm, rotated rx -179.9 ry 0 rz -90 deg; joints [37.178, -72.233, 112.144, -129.537, 51.571, 143.939]
  MoveL 1770 to (255.65, 30.53, -66.6) mm, rotated rx -179.9 ry 0 rz -90 deg; joints [37.178, -72.233, 112.144, -129.537, 51.571, 143.939]
  MoveL 1771 to (248.97, 30.52, -66.6) mm, rotated rx -179.9 ry 0 rz -90 deg; joints [36.948, -72.474, 112.472, -129.827, 51.492, 144.169]
  MoveC 1772 to (244.46, 30.53, -67.86) mm, rotated rx -179.9 ry 0 rz -90 deg; joints [36.76, -72.574, 112.611, -130.045, 51.406, 144.325] to (241.27, 30.53, -71.28) mm, rotated rx -179.9 ry 0 rz -90 deg; joints [36.561, -72.522, 112.546, -130.244, 51.281, 144.438]
  MoveL 1773 to (241.27, 30.52, -71.28) mm, rotated rx -179.9 ry 0 rz -90 deg; joints [36.561, -72.522, 112.546, -130.244, 51.281, 144.438]
  MoveC 1774 to (238.08, 30.52, -74.7) mm, rotated rx -179.9 ry 0 rz -90 deg; joints [36.362, -72.469, 112.479, -130.442, 51.157, 144.551] to (233.58, 30.52, -75.96) mm, rotated rx -179.9 ry 0 rz -90 deg; joints [36.173, -72.567, 112.614, -130.663, 51.071, 144.709]
  MoveL 1775 to (233.58, 30.53, -75.96) mm, rotated rx -179.9 ry 0 rz -90 deg; joints [36.173, -72.567, 112.614, -130.663, 51.071, 144.709]
  MoveL 1776 to (-246.29, 30.53, -75.96) mm, rotated rx -179.9 ry 0 rz -90 deg; joints [15.8, -85.689, 128.839, -157.156, 44.517, 163.757]
  MoveC 1777 to (-249.01, 30.53, -77.09) mm, rotated rx -179.9 ry 0 rz -90 deg; joints [15.649, -85.666, 128.816, -157.363, 44.474, 163.902] to (-250.14, 30.53, -79.82) mm, rotated rx -179.9 ry 0 rz -90 deg; joints [15.555, -85.515, 128.654, -157.488, 44.439, 163.987]
  MoveL 1778 to (-250.14, 30.52, -79.82) mm, rotated rx -179.9 ry 0 rz -90 deg; joints [15.555, -85.515, 128.654, -157.488, 44.439, 163.987]
  MoveL 1779 to (-250.14, 30.52, -232.42) mm, rotated rx -179.9 ry 0 rz -90 deg; joints [13.686, -76.26, 117.832, -159.498, 42.475, 165.02]
  MoveC 1780 to (-249.01, 30.53, -235.14) mm, rotated rx -179.9 ry 0 rz -90 deg; joints [13.706, -76.082, 117.608, -159.45, 42.436, 164.975] to (-246.29, 30.52, -236.27) mm, rotated rx -179.9 ry 0 rz -90 deg; joints [13.814, -75.977, 117.472, -159.285, 42.436, 164.847]
  MoveL 1781 to (-246.29, 30.52, -236.27) mm, rotated rx -179.9 ry 0 rz -90 deg; joints [13.814, -75.977, 117.472, -159.285, 42.436, 164.847]
  MoveL 1782 to (246.29, 30.53, -236.27) mm, rotated rx -179.9 ry 0 rz -90 deg; joints [32.864, -64.161, 100.818, -131.994, 46.883, 143.607]
  MoveC 1783 to (249.01, 30.53, -235.14) mm, rotated rx -179.9 ry 0 rz -90 deg; joints [32.977, -64.129, 100.768, -131.857, 46.939, 143.505] to (250.14, 30.53, -232.42) mm, rotated rx -179.9 ry 0 rz -90 deg; joints [33.072, -64.231, 100.917, -131.785, 47.027, 143.483]
  MoveL 1784 to (250.14, 30.52, -232.42) mm, rotated rx -179.9 ry 0 rz -90 deg; joints [33.072, -64.231, 100.917, -131.785, 47.027, 143.483]
  MoveL 1785 to (250.14, 30.52, -79.82) mm, rotated rx -179.9 ry 0 rz -90 deg; joints [36.647, -71.793, 111.562, -129.998, 51.168, 144.133]
  MoveC 1786 to (249.01, 30.52, -77.09) mm, rotated rx -179.9 ry 0 rz -90 deg; joints [36.679, -71.965, 111.794, -130.002, 51.225, 144.172] to (246.29, 30.52, -75.96) mm, rotated rx -179.9 ry 0 rz -90 deg; joints [36.614, -72.117, 112, -130.103, 51.222, 144.267]
  MoveL 1787 to (246.29, 30.53, -75.96) mm, rotated rx -179.9 ry 0 rz -90 deg; joints [36.614, -72.117, 112, -130.103, 51.222, 144.267]
  MoveL 1788 to (233.58, 30.53, -75.96) mm, rotated rx -179.9 ry 0 rz -90 deg; joints [36.173, -72.567, 112.614, -130.663, 51.071, 144.709]
  MoveC 1789 to (229.36, 30.53, -77.24) mm, rotated rx -179.9 ry 0 rz -90 deg; joints [35.994, -72.653, 112.734, -130.872, 50.989, 144.857] to (226.56, 30.52, -80.65) mm, rotated rx -179.9 ry 0 rz -90 deg; joints [35.809, -72.584, 112.646, -131.054, 50.87, 144.957]
  MoveL 1790 to (226.56, 30.53, -80.65) mm, rotated rx -179.9 ry 0 rz -90 deg; joints [35.809, -72.584, 112.646, -131.054, 50.87, 144.957]
  MoveC 1791 to (223.75, 30.53, -84.05) mm, rotated rx -179.9 ry 0 rz -90 deg; joints [35.625, -72.515, 112.558, -131.236, 50.751, 145.058] to (219.54, 30.53, -85.33) mm, rotated rx -179.9 ry 0 rz -90 deg; joints [35.444, -72.599, 112.674, -131.447, 50.669, 145.208]
  MoveL 1792 to (219.54, 30.53, -85.33) mm, rotated rx -179.9 ry 0 rz -90 deg; joints [35.444, -72.599, 112.674, -131.447, 50.669, 145.208]
  MoveL 1793 to (-236.92, 30.53, -85.33) mm, rotated rx -179.9 ry 0 rz -90 deg; joints [16.129, -84.94, 128.025, -156.681, 44.551, 163.406]
  MoveC 1794 to (-239.65, 30.53, -86.46) mm, rotated rx -179.9 ry 0 rz -90 deg; joints [15.979, -84.918, 128.003, -156.885, 44.508, 163.549] to (-240.78, 30.52, -89.18) mm, rotated rx -179.9 ry 0 rz -90 deg; joints [15.886, -84.769, 127.841, -157.009, 44.47, 163.632]
  MoveL 1795 to (-240.78, 30.53, -89.18) mm, rotated rx -179.9 ry 0 rz -90 deg; joints [15.886, -84.769, 127.841, -157.009, 44.47, 163.632]
  MoveL 1796 to (-240.78, 30.52, -223.05) mm, rotated rx -179.9 ry 0 rz -90 deg; joints [14.203, -76.678, 118.353, -158.801, 42.708, 164.54]
  MoveC 1797 to (-239.65, 30.52, -225.78) mm, rotated rx -179.9 ry 0 rz -90 deg; joints [14.222, -76.5, 118.129, -158.755, 42.67, 164.496] to (-236.92, 30.52, -226.91) mm, rotated rx -179.9 ry 0 rz -90 deg; joints [14.33, -76.393, 117.992, -158.591, 42.672, 164.37]
  MoveL 1798 to (-236.92, 30.52, -226.91) mm, rotated rx -179.9 ry 0 rz -90 deg; joints [14.33, -76.393, 117.992, -158.591, 42.672, 164.37]
  MoveL 1799 to (236.92, 30.52, -226.91) mm, rotated rx -179.9 ry 0 rz -90 deg; joints [32.755, -64.944, 101.976, -132.374, 47.071, 144.067]
  MoveC 1800 to (239.65, 30.53, -225.78) mm, rotated rx -179.9 ry 0 rz -90 deg; joints [32.869, -64.912, 101.927, -132.236, 47.127, 143.966] to (240.78, 30.53, -223.05) mm, rotated rx -179.9 ry 0 rz -90 deg; joints [32.965, -65.014, 102.075, -132.161, 47.214, 143.942]
  MoveL 1801 to (240.78, 30.53, -223.05) mm, rotated rx -179.9 ry 0 rz -90 deg; joints [32.965, -65.014, 102.075, -132.161, 47.214, 143.942]
  MoveL 1802 to (240.78, 30.52, -89.18) mm, rotated rx -179.9 ry 0 rz -90 deg; joints [36.087, -71.669, 111.407, -130.562, 50.82, 144.461]
  MoveC 1803 to (239.65, 30.53, -86.46) mm, rotated rx -179.9 ry 0 rz -90 deg; joints [36.117, -71.842, 111.64, -130.568, 50.876, 144.501] to (236.92, 30.53, -85.33) mm, rotated rx -179.9 ry 0 rz -90 deg; joints [36.052, -71.992, 111.845, -130.671, 50.874, 144.597]
  MoveL 1804 to (236.92, 30.53, -85.33) mm, rotated rx -179.9 ry 0 rz -90 deg; joints [36.052, -71.992, 111.845, -130.671, 50.874, 144.597]
  MoveL 1805 to (219.54, 30.53, -85.33) mm, rotated rx -179.9 ry 0 rz -90 deg; joints [35.444, -72.599, 112.674, -131.447, 50.669, 145.208]
  MoveC 1806 to (215.32, 30.52, -86.61) mm, rotated rx -179.9 ry 0 rz -90 deg; joints [35.264, -72.682, 112.789, -131.658, 50.586, 145.357] to (212.51, 30.53, -90.01) mm, rotated rx -179.9 ry 0 rz -90 deg; joints [35.08, -72.61, 112.697, -131.842, 50.468, 145.459]
  MoveL 1807 to (212.51, 30.53, -90.01) mm, rotated rx -179.9 ry 0 rz -90 deg; joints [35.08, -72.61, 112.697, -131.842, 50.468, 145.459]
  MoveC 1808 to (209.71, 30.53, -93.41) mm, rotated rx -179.9 ry 0 rz -90 deg; joints [34.896, -72.537, 112.604, -132.025, 50.35, 145.562] to (205.49, 30.52, -94.69) mm, rotated rx -179.9 ry 0 rz -90 deg; joints [34.715, -72.618, 112.716, -132.238, 50.268, 145.713]
  MoveL 1809 to (205.49, 30.52, -94.69) mm, rotated rx -179.9 ry 0 rz -90 deg; joints [34.715, -72.618, 112.716, -132.238, 50.268, 145.713]
  MoveL 1810 to (-227.56, 30.52, -94.69) mm, rotated rx -179.9 ry 0 rz -90 deg; joints [16.451, -84.194, 127.203, -156.212, 44.575, 163.055]
  MoveC 1811 to (-230.29, 30.52, -95.82) mm, rotated rx -179.9 ry 0 rz -90 deg; joints [16.303, -84.173, 127.181, -156.413, 44.532, 163.196] to (-231.41, 30.52, -98.54) mm, rotated rx -179.9 ry 0 rz -90 deg; joints [16.209, -84.025, 127.019, -156.535, 44.491, 163.277]
  MoveL 1812 to (-231.41, 30.53, -98.54) mm, rotated rx -179.9 ry 0 rz -90 deg; joints [16.209, -84.025, 127.019, -156.535, 44.491, 163.277]
  MoveL 1813 to (-231.41, 30.52, -213.69) mm, rotated rx -179.9 ry 0 rz -90 deg; joints [14.726, -77.091, 118.863, -158.1, 42.942, 164.059]
  MoveC 1814 to (-230.29, 30.52, -216.42) mm, rotated rx -179.9 ry 0 rz -90 deg; joints [14.744, -76.912, 118.64, -158.057, 42.905, 164.016] to (-227.56, 30.53, -217.54) mm, rotated rx -179.9 ry 0 rz -90 deg; joints [14.851, -76.804, 118.502, -157.894, 42.908, 163.891]
  MoveL 1815 to (-227.56, 30.53, -217.55) mm, rotated rx -179.9 ry 0 rz -90 deg; joints [14.851, -76.804, 118.502, -157.894, 42.908, 163.891]
  MoveL 1816 to (227.56, 30.53, -217.55) mm, rotated rx -179.9 ry 0 rz -90 deg; joints [32.644, -65.724, 103.121, -132.745, 47.252, 144.515]
  MoveC 1817 to (230.29, 30.53, -216.42) mm, rotated rx -179.9 ry 0 rz -90 deg; joints [32.759, -65.693, 103.073, -132.606, 47.309, 144.414] to (231.41, 30.52, -213.69) mm, rotated rx -179.9 ry 0 rz -90 deg; joints [32.856, -65.795, 103.219, -132.53, 47.395, 144.387]
  MoveL 1818 to (231.41, 30.53, -213.69) mm, rotated rx -179.9 ry 0 rz -90 deg; joints [32.856, -65.795, 103.219, -132.53, 47.395, 144.387]
  MoveL 1819 to (231.41, 30.52, -98.54) mm, rotated rx -179.9 ry 0 rz -90 deg; joints [35.529, -71.538, 111.242, -131.128, 50.473, 144.791]
  MoveC 1820 to (230.29, 30.53, -95.82) mm, rotated rx -179.9 ry 0 rz -90 deg; joints [35.558, -71.711, 111.476, -131.136, 50.529, 144.832] to (227.56, 30.52, -94.69) mm, rotated rx -179.9 ry 0 rz -90 deg; joints [35.491, -71.86, 111.68, -131.24, 50.527, 144.929]
  MoveL 1821 to (227.56, 30.53, -94.69) mm, rotated rx -179.9 ry 0 rz -90 deg; joints [35.491, -71.86, 111.68, -131.24, 50.527, 144.929]
  MoveL 1822 to (205.49, 30.52, -94.69) mm, rotated rx -179.9 ry 0 rz -90 deg; joints [34.715, -72.618, 112.716, -132.238, 50.268, 145.713]
  MoveC 1823 to (201.27, 30.52, -95.97) mm, rotated rx -179.9 ry 0 rz -90 deg; joints [34.533, -72.698, 112.827, -132.452, 50.186, 145.864] to (198.47, 30.52, -99.37) mm, rotated rx -179.9 ry 0 rz -90 deg; joints [34.35, -72.623, 112.731, -132.637, 50.069, 145.967]
  MoveL 1824 to (198.47, 30.52, -99.37) mm, rotated rx -179.9 ry 0 rz -90 deg; joints [34.35, -72.623, 112.731, -132.637, 50.069, 145.967]
  MoveC 1825 to (195.67, 30.52, -102.78) mm, rotated rx -179.9 ry 0 rz -90 deg; joints [34.167, -72.547, 112.633, -132.821, 49.951, 146.071] to (191.45, 30.52, -104.05) mm, rotated rx -179.9 ry 0 rz -90 deg; joints [33.985, -72.624, 112.741, -133.037, 49.87, 146.224]
  MoveL 1826 to (191.45, 30.52, -104.05) mm, rotated rx -179.9 ry 0 rz -90 deg; joints [33.985, -72.624, 112.741, -133.037, 49.87, 146.224]
  MoveL 1827 to (-218.2, 30.53, -104.05) mm, rotated rx -179.9 ry 0 rz -90 deg; joints [16.766, -83.451, 126.371, -155.747, 44.589, 162.704]
  MoveC 1828 to (-220.92, 30.52, -105.18) mm, rotated rx -179.9 ry 0 rz -90 deg; joints [16.62, -83.431, 126.351, -155.946, 44.545, 162.844] to (-222.05, 30.53, -107.91) mm, rotated rx -179.9 ry 0 rz -90 deg; joints [16.527, -83.285, 126.189, -156.065, 44.502, 162.923]
  MoveL 1829 to (-222.05, 30.53, -107.91) mm, rotated rx -179.9 ry 0 rz -90 deg; joints [16.527, -83.285, 126.189, -156.065, 44.502, 162.923]
  MoveL 1830 to (-222.05, 30.53, -204.33) mm, rotated rx -179.9 ry 0 rz -90 deg; joints [15.254, -77.498, 119.363, -157.395, 43.176, 163.577]
  MoveC 1831 to (-220.92, 30.52, -207.05) mm, rotated rx -179.9 ry 0 rz -90 deg; joints [15.271, -77.319, 119.14, -157.354, 43.141, 163.535] to (-218.2, 30.52, -208.18) mm, rotated rx -179.9 ry 0 rz -90 deg; joints [15.378, -77.209, 119.001, -157.192, 43.145, 163.412]
  MoveL 1832 to (-218.2, 30.53, -208.18) mm, rotated rx -179.9 ry 0 rz -90 deg; joints [15.378, -77.209, 119.001, -157.192, 43.145, 163.412]
  MoveL 1833 to (218.2, 30.53, -208.18) mm, rotated rx -179.9 ry 0 rz -90 deg; joints [32.531, -66.502, 104.253, -133.109, 47.428, 144.95]
  MoveC 1834 to (220.92, 30.52, -207.05) mm, rotated rx -179.9 ry 0 rz -90 deg; joints [32.647, -66.472, 104.206, -132.969, 47.484, 144.849] to (222.05, 30.52, -204.33) mm, rotated rx -179.9 ry 0 rz -90 deg; joints [32.745, -66.574, 104.351, -132.89, 47.57, 144.82]
  MoveL 1835 to (222.05, 30.53, -204.33) mm, rotated rx -179.9 ry 0 rz -90 deg; joints [32.745, -66.574, 104.351, -132.89, 47.57, 144.82]
  MoveL 1836 to (222.05, 30.52, -107.91) mm, rotated rx -179.9 ry 0 rz -90 deg; joints [34.973, -71.399, 111.066, -131.696, 50.127, 145.123]
  MoveC 1837 to (220.92, 30.52, -105.18) mm, rotated rx -179.9 ry 0 rz -90 deg; joints [35, -71.572, 111.301, -131.705, 50.184, 145.165] to (218.2, 30.52, -104.05) mm, rotated rx -179.9 ry 0 rz -90 deg; joints [34.932, -71.721, 111.504, -131.811, 50.181, 145.263]
  MoveL 1838 to (218.2, 30.52, -104.05) mm, rotated rx -179.9 ry 0 rz -90 deg; joints [34.932, -71.721, 111.504, -131.811, 50.181, 145.263]
  MoveL 1839 to (191.45, 30.52, -104.05) mm, rotated rx -179.9 ry 0 rz -90 deg; joints [33.985, -72.624, 112.741, -133.037, 49.87, 146.224]
  MoveC 1840 to (187.23, 30.53, -105.33) mm, rotated rx -179.9 ry 0 rz -90 deg; joints [33.802, -72.701, 112.847, -133.253, 49.788, 146.377] to (184.43, 30.52, -108.73) mm, rotated rx -179.9 ry 0 rz -90 deg; joints [33.62, -72.623, 112.747, -133.438, 49.672, 146.481]
  MoveL 1841 to (184.43, 30.53, -108.73) mm, rotated rx -179.9 ry 0 rz -90 deg; joints [33.62, -72.623, 112.747, -133.438, 49.672, 146.481]
  MoveC 1842 to (181.62, 30.53, -112.14) mm, rotated rx -179.9 ry 0 rz -90 deg; joints [33.437, -72.544, 112.645, -133.623, 49.555, 146.586] to (177.4, 30.53, -113.42) mm, rotated rx -179.9 ry 0 rz -90 deg; joints [33.254, -72.618, 112.748, -133.842, 49.474, 146.74]
  MoveL 1843 to (177.4, 30.53, -113.42) mm, rotated rx -179.9 ry 0 rz -90 deg; joints [33.254, -72.618, 112.748, -133.842, 49.474, 146.74]
  MoveL 1844 to (-208.84, 30.52, -113.42) mm, rotated rx -179.9 ry 0 rz -90 deg; joints [17.075, -82.71, 125.532, -155.286, 44.593, 162.352]
  MoveC 1845 to (-211.56, 30.52, -114.54) mm, rotated rx -179.9 ry 0 rz -90 deg; joints [16.93, -82.691, 125.513, -155.483, 44.548, 162.49] to (-212.69, 30.52, -117.27) mm, rotated rx -179.9 ry 0 rz -90 deg; joints [16.837, -82.546, 125.349, -155.601, 44.503, 162.567]
  MoveL 1846 to (-212.69, 30.52, -117.27) mm, rotated rx -179.9 ry 0 rz -90 deg; joints [16.837, -82.546, 125.349, -155.601, 44.503, 162.567]
  MoveL 1847 to (-212.69, 30.52, -194.97) mm, rotated rx -179.9 ry 0 rz -90 deg; joints [15.788, -77.9, 119.852, -156.687, 43.412, 163.093]
  MoveC 1848 to (-211.56, 30.52, -197.69) mm, rotated rx -179.9 ry 0 rz -90 deg; joints [15.803, -77.72, 119.63, -156.647, 43.378, 163.053] to (-208.84, 30.52, -198.82) mm, rotated rx -179.9 ry 0 rz -90 deg; joints [15.91, -77.608, 119.491, -156.487, 43.384, 162.931]
  MoveL 1849 to (-208.84, 30.52, -198.82) mm, rotated rx -179.9 ry 0 rz -90 deg; joints [15.91, -77.608, 119.491, -156.487, 43.384, 162.931]
  MoveL 1850 to (208.84, 30.53, -198.82) mm, rotated rx -179.9 ry 0 rz -90 deg; joints [32.416, -67.279, 105.372, -133.465, 47.597, 145.373]
  MoveC 1851 to (211.56, 30.52, -197.69) mm, rotated rx -179.9 ry 0 rz -90 deg; joints [32.533, -67.249, 105.327, -133.324, 47.653, 145.272] to (212.69, 30.53, -194.97) mm, rotated rx -179.9 ry 0 rz -90 deg; joints [32.632, -67.351, 105.471, -133.243, 47.738, 145.241]
  MoveL 1852 to (212.69, 30.53, -194.97) mm, rotated rx -179.9 ry 0 rz -90 deg; joints [32.632, -67.351, 105.471, -133.243, 47.738, 145.241]
  MoveL 1853 to (212.69, 30.53, -117.27) mm, rotated rx -179.9 ry 0 rz -90 deg; joints [34.418, -71.253, 110.88, -132.264, 49.783, 145.457]
  MoveC 1854 to (211.56, 30.53, -114.54) mm, rotated rx -179.9 ry 0 rz -90 deg; joints [34.444, -71.426, 111.115, -132.275, 49.839, 145.5] to (208.84, 30.53, -113.42) mm, rotated rx -179.9 ry 0 rz -90 deg; joints [34.376, -71.574, 111.318, -132.383, 49.837, 145.599]
  MoveL 1855 to (208.84, 30.52, -113.42) mm, rotated rx -179.9 ry 0 rz -90 deg; joints [34.376, -71.574, 111.318, -132.383, 49.837, 145.599]
  MoveL 1856 to (177.4, 30.53, -113.42) mm, rotated rx -179.9 ry 0 rz -90 deg; joints [33.254, -72.618, 112.748, -133.842, 49.474, 146.74]
  MoveC 1857 to (173.18, 30.52, -114.69) mm, rotated rx -179.9 ry 0 rz -90 deg; joints [33.071, -72.691, 112.85, -134.06, 49.393, 146.895] to (170.38, 30.52, -118.1) mm, rotated rx -179.9 ry 0 rz -90 deg; joints [32.889, -72.61, 112.745, -134.247, 49.277, 147.001]
  MoveL 1858 to (170.38, 30.52, -118.1) mm, rotated rx -179.9 ry 0 rz -90 deg; joints [32.889, -72.61, 112.745, -134.247, 49.277, 147.001]
  MoveC 1859 to (167.58, 30.53, -121.5) mm, rotated rx -179.9 ry 0 rz -90 deg; joints [32.708, -72.527, 112.639, -134.433, 49.161, 147.107] to (163.36, 30.52, -122.78) mm, rotated rx -179.9 ry 0 rz -90 deg; joints [32.524, -72.598, 112.738, -134.653, 49.081, 147.263]
  MoveL 1860 to (163.36, 30.53, -122.78) mm, rotated rx -179.9 ry 0 rz -90 deg; joints [32.524, -72.598, 112.738, -134.653, 49.081, 147.263]
  MoveL 1861 to (-199.47, 30.52, -122.78) mm, rotated rx -179.9 ry 0 rz -90 deg; joints [17.378, -81.971, 124.683, -154.829, 44.587, 161.999]
  MoveC 1862 to (-202.2, 30.52, -123.91) mm, rotated rx -179.9 ry 0 rz -90 deg; joints [17.234, -81.953, 124.665, -155.023, 44.542, 162.135] to (-203.33, 30.52, -126.63) mm, rotated rx -179.9 ry 0 rz -90 deg; joints [17.142, -81.81, 124.501, -155.139, 44.495, 162.21]
  MoveL 1863 to (-203.33, 30.52, -126.63) mm, rotated rx -179.9 ry 0 rz -90 deg; joints [17.142, -81.81, 124.501, -155.139, 44.495, 162.21]
  MoveL 1864 to (-203.33, 30.52, -185.6) mm, rotated rx -179.9 ry 0 rz -90 deg; joints [16.327, -78.296, 120.331, -155.975, 43.649, 162.609]
  MoveC 1865 to (-202.2, 30.52, -188.33) mm, rotated rx -179.9 ry 0 rz -90 deg; joints [16.342, -78.115, 120.11, -155.937, 43.616, 162.57] to (-199.47, 30.52, -189.46) mm, rotated rx -179.9 ry 0 rz -90 deg; joints [16.448, -78.002, 119.969, -155.778, 43.623, 162.449]
  MoveL 1866 to (-199.47, 30.52, -189.46) mm, rotated rx -179.9 ry 0 rz -90 deg; joints [16.448, -78.002, 119.969, -155.778, 43.623, 162.449]
  MoveL 1867 to (199.47, 30.53, -189.46) mm, rotated rx -179.9 ry 0 rz -90 deg; joints [32.299, -68.054, 106.48, -133.815, 47.759, 145.784]
  MoveC 1868 to (202.2, 30.53, -188.33) mm, rotated rx -179.9 ry 0 rz -90 deg; joints [32.417, -68.025, 106.435, -133.672, 47.816, 145.683] to (203.33, 30.52, -185.6) mm, rotated rx -179.9 ry 0 rz -90 deg; joints [32.516, -68.127, 106.578, -133.589, 47.9, 145.65]
  MoveL 1869 to (203.33, 30.52, -185.6) mm, rotated rx -179.9 ry 0 rz -90 deg; joints [32.516, -68.127, 106.578, -133.589, 47.9, 145.65]
  MoveL 1870 to (203.33, 30.52, -126.63) mm, rotated rx -179.9 ry 0 rz -90 deg; joints [33.865, -71.099, 110.682, -132.834, 49.44, 145.793]
  MoveC 1871 to (202.2, 30.53, -123.91) mm, rotated rx -179.9 ry 0 rz -90 deg; joints [33.89, -71.273, 110.919, -132.847, 49.496, 145.837] to (199.47, 30.52, -122.78) mm, rotated rx -179.9 ry 0 rz -90 deg; joints [33.821, -71.42, 111.12, -132.956, 49.494, 145.937]
  MoveL 1872 to (199.47, 30.52, -122.78) mm, rotated rx -179.9 ry 0 rz -90 deg; joints [33.821, -71.42, 111.12, -132.956, 49.494, 145.937]
  MoveL 1873 to (163.36, 30.53, -122.78) mm, rotated rx -179.9 ry 0 rz -90 deg; joints [32.524, -72.598, 112.738, -134.653, 49.081, 147.263]
  MoveC 1874 to (159.14, 30.53, -124.06) mm, rotated rx -179.9 ry 0 rz -90 deg; joints [32.341, -72.668, 112.836, -134.874, 49, 147.42] to (156.34, 30.52, -127.46) mm, rotated rx -179.9 ry 0 rz -90 deg; joints [32.159, -72.584, 112.727, -135.061, 48.885, 147.527]
  MoveL 1875 to (156.34, 30.52, -127.46) mm, rotated rx -179.9 ry 0 rz -90 deg; joints [32.159, -72.584, 112.727, -135.061, 48.885, 147.527]
  MoveC 1876 to (153.54, 30.52, -130.86) mm, rotated rx -179.9 ry 0 rz -90 deg; joints [31.979, -72.498, 112.616, -135.248, 48.77, 147.634] to (149.32, 30.52, -132.14) mm, rotated rx -179.9 ry 0 rz -90 deg; joints [31.795, -72.566, 112.711, -135.471, 48.69, 147.792]
  MoveL 1877 to (149.32, 30.52, -132.14) mm, rotated rx -179.9 ry 0 rz -90 deg; joints [31.795, -72.566, 112.711, -135.471, 48.69, 147.792]
  MoveL 1878 to (-190.11, 30.53, -132.14) mm, rotated rx -179.9 ry 0 rz -90 deg; joints [17.675, -81.234, 123.826, -154.375, 44.572, 161.644]
  MoveC 1879 to (-192.84, 30.53, -133.27) mm, rotated rx -179.9 ry 0 rz -90 deg; joints [17.532, -81.218, 123.809, -154.567, 44.526, 161.779] to (-193.96, 30.53, -135.99) mm, rotated rx -179.9 ry 0 rz -90 deg; joints [17.44, -81.076, 123.644, -154.682, 44.477, 161.852]
  MoveL 1880 to (-193.96, 30.52, -135.99) mm, rotated rx -179.9 ry 0 rz -90 deg; joints [17.44, -81.076, 123.644, -154.682, 44.477, 161.852]
  MoveL 1881 to (-193.96, 30.52, -176.24) mm, rotated rx -179.9 ry 0 rz -90 deg; joints [16.872, -78.686, 120.8, -155.259, 43.888, 162.123]
  MoveC 1882 to (-192.84, 30.52, -178.97) mm, rotated rx -179.9 ry 0 rz -90 deg; joints [16.885, -78.505, 120.579, -155.223, 43.856, 162.086] to (-190.11, 30.52, -180.09) mm, rotated rx -179.9 ry 0 rz -90 deg; joints [16.992, -78.39, 120.438, -155.065, 43.864, 161.966]
  MoveL 1883 to (-190.11, 30.52, -180.09) mm, rotated rx -179.9 ry 0 rz -90 deg; joints [16.992, -78.39, 120.438, -155.065, 43.864, 161.966]
  MoveL 1884 to (190.11, 30.53, -180.09) mm, rotated rx -179.9 ry 0 rz -90 deg; joints [32.179, -68.829, 107.576, -134.157, 47.915, 146.184]
  MoveC 1885 to (192.84, 30.53, -178.97) mm, rotated rx -179.9 ry 0 rz -90 deg; joints [32.299, -68.8, 107.532, -134.014, 47.973, 146.082] to (193.96, 30.52, -176.24) mm, rotated rx -179.9 ry 0 rz -90 deg; joints [32.399, -68.902, 107.674, -133.928, 48.056, 146.047]
  MoveL 1886 to (193.96, 30.53, -176.24) mm, rotated rx -179.9 ry 0 rz -90 deg; joints [32.399, -68.902, 107.674, -133.928, 48.056, 146.047]
  MoveL 1887 to (193.96, 30.53, -135.99) mm, rotated rx -179.9 ry 0 rz -90 deg; joints [33.315, -70.938, 110.474, -133.406, 49.098, 146.131]
  MoveC 1888 to (192.84, 30.52, -133.27) mm, rotated rx -179.9 ry 0 rz -90 deg; joints [33.338, -71.112, 110.712, -133.419, 49.155, 146.175] to (190.11, 30.53, -132.14) mm, rotated rx -179.9 ry 0 rz -90 deg; joints [33.268, -71.258, 110.912, -133.531, 49.153, 146.277]
  MoveL 1889 to (190.11, 30.52, -132.14) mm, rotated rx -179.9 ry 0 rz -90 deg; joints [33.268, -71.258, 110.912, -133.531, 49.153, 146.277]
  MoveL 1890 to (149.32, 30.52, -132.14) mm, rotated rx -179.9 ry 0 rz -90 deg; joints [31.795, -72.566, 112.711, -135.471, 48.69, 147.792]
  MoveC 1891 to (145.1, 30.52, -133.42) mm, rotated rx -179.9 ry 0 rz -90 deg; joints [31.61, -72.633, 112.804, -135.695, 48.61, 147.951] to (142.29, 30.52, -136.82) mm, rotated rx -179.9 ry 0 rz -90 deg; joints [31.43, -72.545, 112.69, -135.883, 48.496, 148.058]
  MoveL 1892 to (142.29, 30.53, -136.82) mm, rotated rx -179.9 ry 0 rz -90 deg; joints [31.43, -72.545, 112.69, -135.883, 48.496, 148.058]
  MoveC 1893 to (139.49, 30.53, -140.23) mm, rotated rx -179.9 ry 0 rz -90 deg; joints [31.25, -72.457, 112.576, -136.07, 48.381, 148.166] to (135.27, 30.53, -141.5) mm, rotated rx -179.9 ry 0 rz -90 deg; joints [31.066, -72.521, 112.666, -136.296, 48.302, 148.326]
  MoveL 1894 to (135.27, 30.52, -141.5) mm, rotated rx -179.9 ry 0 rz -90 deg; joints [31.066, -72.521, 112.666, -136.296, 48.302, 148.326]
  MoveL 1895 to (-180.75, 30.52, -141.5) mm, rotated rx -179.9 ry 0 rz -90 deg; joints [17.966, -80.5, 122.96, -153.924, 44.547, 161.288]
  MoveC 1896 to (-183.47, 30.53, -142.63) mm, rotated rx -179.9 ry 0 rz -90 deg; joints [17.825, -80.484, 122.943, -154.114, 44.501, 161.421] to (-184.6, 30.53, -145.36) mm, rotated rx -179.9 ry 0 rz -90 deg; joints [17.733, -80.344, 122.778, -154.227, 44.449, 161.492]
  MoveL 1897 to (-184.6, 30.52, -145.36) mm, rotated rx -179.9 ry 0 rz -90 deg; joints [17.733, -80.344, 122.778, -154.227, 44.449, 161.492]
  MoveL 1898 to (-184.6, 30.52, -166.88) mm, rotated rx -179.9 ry 0 rz -90 deg; joints [17.423, -79.07, 121.258, -154.539, 44.128, 161.636]
  MoveC 1899 to (-183.47, 30.52, -169.6) mm, rotated rx -179.9 ry 0 rz -90 deg; joints [17.435, -78.889, 121.038, -154.505, 44.097, 161.601] to (-180.75, 30.52, -170.73) mm, rotated rx -179.9 ry 0 rz -90 deg; joints [17.541, -78.772, 120.896, -154.349, 44.107, 161.482]
  MoveL 1900 to (-180.75, 30.52, -170.73) mm, rotated rx -179.9 ry 0 rz -90 deg; joints [17.541, -78.772, 120.896, -154.349, 44.107, 161.482]
  MoveL 1901 to (180.75, 30.53, -170.73) mm, rotated rx -179.9 ry 0 rz -90 deg; joints [32.058, -69.602, 108.66, -134.493, 48.065, 146.572]
  MoveC 1902 to (183.47, 30.52, -169.6) mm, rotated rx -179.9 ry 0 rz -90 deg; joints [32.179, -69.574, 108.617, -134.349, 48.122, 146.47] to (184.6, 30.52, -166.88) mm, rotated rx -179.9 ry 0 rz -90 deg; joints [32.279, -69.676, 108.758, -134.261, 48.205, 146.433]
  MoveL 1903 to (184.6, 30.53, -166.88) mm, rotated rx -179.9 ry 0 rz -90 deg; joints [32.279, -69.676, 108.758, -134.261, 48.205, 146.433]
  MoveL 1904 to (184.6, 30.52, -145.36) mm, rotated rx -179.9 ry 0 rz -90 deg; joints [32.766, -70.769, 110.256, -133.978, 48.757, 146.471]
  MoveC 1905 to (183.47, 30.52, -142.63) mm, rotated rx -179.9 ry 0 rz -90 deg; joints [32.789, -70.943, 110.494, -133.993, 48.814, 146.516] to (180.75, 30.53, -141.5) mm, rotated rx -179.9 ry 0 rz -90 deg; joints [32.718, -71.088, 110.693, -134.106, 48.813, 146.619]
  MoveL 1906 to (180.75, 30.52, -141.5) mm, rotated rx -179.9 ry 0 rz -90 deg; joints [32.718, -71.088, 110.693, -134.106, 48.813, 146.619]
  MoveL 1907 to (135.27, 30.52, -141.5) mm, rotated rx -179.9 ry 0 rz -90 deg; joints [31.066, -72.521, 112.666, -136.296, 48.302, 148.326]
  MoveC 1908 to (131.05, 30.53, -142.78) mm, rotated rx -179.9 ry 0 rz -90 deg; joints [30.881, -72.584, 112.755, -136.522, 48.223, 148.487] to (128.25, 30.53, -146.18) mm, rotated rx -179.9 ry 0 rz -90 deg; joints [30.701, -72.493, 112.637, -136.71, 48.109, 148.596]
  MoveL 1909 to (128.25, 30.52, -146.18) mm, rotated rx -179.9 ry 0 rz -90 deg; joints [30.701, -72.493, 112.637, -136.71, 48.109, 148.596]
  MoveC 1910 to (125.45, 30.53, -149.59) mm, rotated rx -179.9 ry 0 rz -90 deg; joints [30.522, -72.402, 112.518, -136.898, 47.996, 148.705] to (121.23, 30.52, -150.87) mm, rotated rx -179.9 ry 0 rz -90 deg; joints [30.337, -72.463, 112.603, -137.126, 47.917, 148.867]
  MoveL 1911 to (121.23, 30.52, -150.87) mm, rotated rx -179.9 ry 0 rz -90 deg; joints [30.337, -72.463, 112.603, -137.126, 47.917, 148.867]
  MoveL 1912 to (-171.39, 30.53, -150.87) mm, rotated rx -179.9 ry 0 rz -90 deg; joints [18.251, -79.767, 122.084, -153.476, 44.513, 160.928]
  MoveC 1913 to (-174.11, 30.52, -151.99) mm, rotated rx -179.9 ry 0 rz -90 deg; joints [18.111, -79.752, 122.069, -153.664, 44.466, 161.06] to (-175.24, 30.53, -154.72) mm, rotated rx -179.9 ry 0 rz -90 deg; joints [18.02, -79.613, 121.904, -153.775, 44.413, 161.13]
  MoveL 1914 to (-175.24, 30.52, -154.72) mm, rotated rx -179.9 ry 0 rz -90 deg; joints [18.02, -79.613, 121.904, -153.775, 44.413, 161.13]
  MoveL 1915 to (-175.24, 30.52, -157.52) mm, rotated rx -179.9 ry 0 rz -90 deg; joints [17.979, -79.448, 121.706, -153.816, 44.37, 161.148]
  MoveC 1916 to (-174.11, 30.53, -160.24) mm, rotated rx -179.9 ry 0 rz -90 deg; joints [17.99, -79.266, 121.487, -153.784, 44.34, 161.115] to (-171.39, 30.52, -161.37) mm, rotated rx -179.9 ry 0 rz -90 deg; joints [18.095, -79.148, 121.343, -153.63, 44.352, 160.998]
  MoveL 1917 to (-171.39, 30.53, -161.37) mm, rotated rx -179.9 ry 0 rz -90 deg; joints [18.095, -79.148, 121.343, -153.63, 44.352, 160.998]
  MoveL 1918 to (171.39, 30.52, -161.37) mm, rotated rx -179.9 ry 0 rz -90 deg; joints [31.934, -70.376, 109.733, -134.823, 48.207, 146.949]
  MoveC 1919 to (174.11, 30.52, -160.24) mm, rotated rx -179.9 ry 0 rz -90 deg; joints [32.056, -70.347, 109.692, -134.678, 48.265, 146.847] to (175.24, 30.53, -157.52) mm, rotated rx -179.9 ry 0 rz -90 deg; joints [32.157, -70.45, 109.832, -134.588, 48.347, 146.808]
  MoveL 1920 to (175.24, 30.52, -157.52) mm, rotated rx -179.9 ry 0 rz -90 deg; joints [32.157, -70.45, 109.832, -134.588, 48.347, 146.808]
  MoveL 1921 to (175.24, 30.52, -154.72) mm, rotated rx -179.9 ry 0 rz -90 deg; joints [32.22, -70.593, 110.026, -134.551, 48.418, 146.812]
  MoveC 1922 to (174.11, 30.53, -151.99) mm, rotated rx -179.9 ry 0 rz -90 deg; joints [32.241, -70.768, 110.265, -134.568, 48.475, 146.858] to (171.39, 30.53, -150.87) mm, rotated rx -179.9 ry 0 rz -90 deg; joints [32.169, -70.912, 110.464, -134.682, 48.474, 146.963]
  MoveL 1923 to (171.39, 30.52, -150.87) mm, rotated rx -179.9 ry 0 rz -90 deg; joints [32.169, -70.912, 110.464, -134.682, 48.474, 146.963]
  MoveL 1924 to (121.23, 30.52, -150.87) mm, rotated rx -179.9 ry 0 rz -90 deg; joints [30.337, -72.463, 112.603, -137.126, 47.917, 148.867]
  MoveL 1925 to (121.01, 30.54, -150.88) mm, rotated rx -179.9 ry 0 rz -90 deg; joints [30.329, -72.469, 112.611, -137.136, 47.913, 148.874]
  MoveL 1926 to (120.8, 30.6, -150.94) mm, rotated rx -179.9 ry 0 rz -90 deg; joints [30.32, -72.474, 112.613, -137.145, 47.907, 148.878]
  MoveL 1927 to (120.62, 30.7, -151.02) mm, rotated rx -179.9 ry 0 rz -90 deg; joints [30.311, -72.479, 112.612, -137.152, 47.898, 148.88]
  MoveL 1928 to (120.47, 30.82, -151.12) mm, rotated rx -179.9 ry 0 rz -90 deg; joints [30.303, -72.483, 112.607, -137.155, 47.888, 148.878]
  MoveL 1929 to (120.35, 30.98, -151.22) mm, rotated rx -179.9 ry 0 rz -90 deg; joints [30.296, -72.486, 112.6, -137.156, 47.876, 148.873]
  MoveL 1930 to (120.26, 31.16, -151.31) mm, rotated rx -179.9 ry 0 rz -90 deg; joints [30.291, -72.49, 112.591, -137.155, 47.864, 148.865]
  MoveL 1931 to (120.2, 31.36, -151.39) mm, rotated rx -179.9 ry 0 rz -90 deg; joints [30.287, -72.495, 112.581, -137.15, 47.852, 148.855]
  MoveL 1932 to (120.17, 31.57, -151.43) mm, rotated rx -179.9 ry 0 rz -90 deg; joints [30.285, -72.501, 112.572, -137.144, 47.84, 148.843]
  MoveL 1933 to (120.16, 31.79, -151.45) mm, rotated rx -179.9 ry 0 rz -90 deg; joints [30.284, -72.508, 112.564, -137.136, 47.828, 148.83]
  Set speed (1000.0 mm/s)
  MoveL 1934 to (120.16, 110.53, -151.45) mm, rotated rx -179.9 ry 0 rz -90 deg; joints [30.245, -74.935, 109.673, -133.558, 44.02, 143.657]
  MoveL 1935 to (315.45, 110.52, -160.95) mm, rotated rx -179.9 ry 0 rz -90 deg; joints [36.758, -67.735, 99.869, -124.573, 46.605, 135.997]
  MoveL 1936 to (315.45, 106.52, -160.95) mm, rotated rx -179.9 ry 0 rz -90 deg; joints [36.76, -67.636, 100.026, -124.769, 46.752, 136.285]
  Set speed (100.0 mm/s)
  MoveL 1937 to (315.45, 58.04, -160.95) mm, rotated rx -179.9 ry 0 rz -90 deg; joints [36.785, -66.344, 101.818, -127.022, 48.578, 139.649]
  MoveL 1938 to (315.47, 57.83, -160.96) mm, rotated rx -179.9 ry 0 rz -90 deg; joints [36.785, -66.337, 101.824, -127.031, 48.586, 139.663]
  MoveL 1939 to (315.51, 57.62, -160.99) mm, rotated rx -179.9 ry 0 rz -90 deg; joints [36.786, -66.328, 101.827, -127.039, 48.593, 139.675]
  MoveL 1940 to (315.58, 57.42, -161.04) mm, rotated rx -179.9 ry 0 rz -90 deg; joints [36.787, -66.317, 101.826, -127.045, 48.6, 139.685]
  MoveL 1941 to (315.68, 57.24, -161.11) mm, rotated rx -179.9 ry 0 rz -90 deg; joints [36.789, -66.305, 101.822, -127.049, 48.606, 139.693]
  MoveL 1942 to (315.81, 57.09, -161.19) mm, rotated rx -179.9 ry 0 rz -90 deg; joints [36.791, -66.292, 101.815, -127.051, 48.611, 139.698]
  MoveL 1943 to (315.96, 56.96, -161.29) mm, rotated rx -179.9 ry 0 rz -90 deg; joints [36.793, -66.278, 101.805, -127.051, 48.615, 139.7]
  MoveL 1944 to (316.12, 56.86, -161.38) mm, rotated rx -179.9 ry 0 rz -90 deg; joints [36.796, -66.264, 101.793, -127.049, 48.618, 139.7]
  MoveL 1945 to (316.31, 56.8, -161.48) mm, rotated rx -179.9 ry 0 rz -90 deg; joints [36.8, -66.251, 101.779, -127.044, 48.619, 139.696]
  MoveL 1946 to (316.5, 56.78, -161.58) mm, rotated rx -179.9 ry 0 rz -90 deg; joints [36.804, -66.239, 101.763, -127.038, 48.62, 139.69]
  MoveL 1947 to (318.61, 56.7, -162.13) mm, rotated rx -179.9 ry 0 rz -90 deg; joints [36.858, -66.132, 101.613, -126.953, 48.629, 139.609]
  MoveL 1948 to (320.79, 56.62, -161.9) mm, rotated rx -179.9 ry 0 rz -90 deg; joints [36.932, -66.062, 101.516, -126.859, 48.661, 139.532]
  MoveL 1949 to (322.74, 56.54, -160.91) mm, rotated rx -179.9 ry 0 rz -90 deg; joints [37.017, -66.037, 101.484, -126.768, 48.712, 139.468]
  MoveL 1950 to (324.2, 56.47, -159.29) mm, rotated rx -179.9 ry 0 rz -90 deg; joints [37.102, -66.061, 101.522, -126.692, 48.776, 139.429]
  MoveL 1951 to (324.99, 56.39, -157.25) mm, rotated rx -179.9 ry 0 rz -90 deg; joints [37.176, -66.129, 101.624, -126.642, 48.845, 139.418]
  MoveL 1952 to (325.01, 56.31, -155.06) mm, rotated rx -179.9 ry 0 rz -90 deg; joints [37.229, -66.233, 101.779, -126.624, 48.91, 139.437]
  MoveL 1953 to (324.24, 56.24, -153.01) mm, rotated rx -179.9 ry 0 rz -90 deg; joints [37.254, -66.359, 101.966, -126.642, 48.963, 139.486]
